REGION Network 4: Block description — Section 3.5 to 3.5
   // ▂▂▂▂▂▂▂▂▂▂▂▂▂▂▂▂▂▂▂▂▂▂▂▂▂▂▂▂▂▂▂▂▂▂▂▂▂▂▂▂▂▂▂▂
   // 3.5     Expressing the calculations in Controller operations
   // 
   // The calculations above must be rendered in a form suitable for the Simatic S7-1500 Controller, 
   // using the mathematical operations available to that Controller, these are listed in Table 2.1.
   // 
   // To perform the calculations in the Controller it will be necessary to use partial calculation to 
   // hold separate components of the overall calculation and combine these to produce the final 
   // result. 
   // 
   // The following sections breakdown each of the response calculations into these partial 
   // calculations and demonstrate how these are then combined to provide a final result that is 
   // compatible with the Controller mathematical operations and Controller notations.
   // 
   // 
   // 
   // ▁▁▁▁▁▁▁▁▁▁▁▁▁▁▁▁▁▁▁▁▁▁▁▁▁▁▁▁▁▁▁▁▁▁▁▁▁▁▁▁▁▁▁▁
   // 3.5.1     Over damped, slow response no overshoot             ζ > 1
   // 
   // 
   // CALCULATION:
   // 
   //       ╓   1 ┌   ζ       ┐   - ω [ ζ ─ √(ζ² ─ 1) ]t       1 ┌   ζ       ┐   - ω [ ζ ┼ √(ζ² ─ 1) ]t ╖
   // y(t) = K║x(t) ─ -- │------------------ ┼ 1│ｅ         ┼ -- │------------------ ─ 1│ｅ           ║
   //       ╙   2 └ √(ζ² ─ 1)     ┘            2 └ √(ζ² ─ 1)     ┘            ╜
   // 
   // 
   // 
   // Is rendered into the correct format as follows:
   // 
   // 
   //  cal_01 = SQRT ( SQR (ζ) - 1)         = √(ζ² ─ 1)
   // 
   //                                  ζ
   //  cal_02 = ζ ÷ cal_01              = -----------------
   //                          √(ζ² ─ 1)
   // 
   //  cal_03 = ζ + cal_01              = ζ ┼ √(ζ² ─ 1)
   // 
   //  cal_04 = -1 × ω × t × cal_03           = - ω [ ζ ┼ √(ζ² ─ 1) ]t
   // 
   //                              -ω [ ζ ┼ √(ζ² ─ 1) ]t 
   //  cal_05 = EXP( cal_04 )              =ｅ
   // 
   //  cal_06 = ζ - cal_01               = ζ ─ √(ζ² ─ 1)
   // 
   //  cal_07 = -1 × ω × t × cal_06           = - ω [ ζ ─ √(ζ² ─ 1) ]t
   // 
   //                            -ω [ ζ ─ √(ζ² ─ 1) ]t 
   //  cal_08 = EXP( cal_07 )              =ｅ
   // 
   //                           1 ┌   ζ       ┐
   //  cal_09 = (cal_02 - 1) × 0.5           = -- │------------------ ─ 1│
   //                           2 └ √(ζ² ─ 1)     ┘
   // 
   //                           1 ┌   ζ       ┐
   //  cal_10 = (cal_02 + 1) × 0.5            = -- │------------------ ┼ 1│
   //                           2 └ √(ζ² ─ 1)     ┘
   // 
   //                           1 ┌   ζ       ┐   -ω [ ζ ┼ √(ζ² ─ 1) ]t
   //  cal_11 = cal_09 × cal_05             = -- │------------------ ─ 1│ｅ
   //                           2 └ √(ζ² ─ 1)     ┘
   // 
   //                           1 ┌   ζ       ┐   -ω [ ζ ─ √(ζ² ─ 1) ]t
   //  cal_12 = cal_10 × cal_08             = -- │------------------ ┼ 1│ｅ
   //                           2 └ √(ζ² ─ 1)     ┘
   // 
   //                          ╓   1 ┌   ζ       ┐   - ω [ ζ ─ √(ζ² ─ 1) ]t       1 ┌   ζ       ┐   - ω [ ζ ┼ √(ζ² ─ 1) ]t ╖
   //  cal_13 = INPUT - cal_12 + cal_11        = ║x(t) ─ -- │------------------ ┼ 1│ｅ         ┼ -- │------------------ ─ 1│ｅ           ║
   //                          ╙   2 └ √(ζ² ─ 1)     ┘            2 └ √(ζ² ─ 1)     ┘            ╜
   // 
   //                             ╓   1 ┌   ζ       ┐   - ω [ ζ ─ √(ζ² ─ 1) ]t       1 ┌   ζ       ┐   - ω [ ζ ┼ √(ζ² ─ 1) ]t ╖
   //  OUTPUT  = K × cal_13             =  K║x(t) ─ -- │------------------ ┼ 1│ｅ         ┼ -- │------------------ ─ 1│ｅ           ║
   //                             ╙   2 └ √(ζ² ─ 1)     ┘            2 └ √(ζ² ─ 1)     ┘            ╜
   // 
   // 
   // 
   // ▁▁▁▁▁▁▁▁▁▁▁▁▁▁▁▁▁▁▁▁▁▁▁▁▁▁▁▁▁▁▁▁▁▁▁▁▁▁▁▁▁▁▁▁
   // 3.5.2     Critically damped, fastest response without overshoot        ζ = 1
   // 
   // 
   // CALCULATION:
   // 
   //       ╓           - ωt  ╖
   // y(t) = K║x(t) ─ (1 ┼ ωt) ｅ  ║
   //       ╙             ╜
   // 
   // 
   // Is rendered into the correct format as follows:
   // 
   // 
   //  cal_01 = -1 × ω × t                = - ωt  
   // 
   //                          - ωt
   //  cal_02 = EXP( cal_01 )              =ｅ
   // 
   //  cal_03 = 1 - cal_01              = 1 ─ (-ωt) = 1 ┼ ωt
   // 
   //                              - ωt
   //  cal_04 = cal_03 × cal_02            = (1 ┼ ωt) ｅ
   // 
   //                                 - ωt
   //  cal_05 = INPUT  - cal_04            = x(t) ─ (1 ┼ ωt) ｅ
   // 
   //                             ╓           - ωt  ╖
   //  OUTPUT  = K × cal_05             =  K║x(t) ─ (1 ┼ ωt) ｅ  ║
   //                             ╙             ╜
   // 
   // 
   // 
   // ▁▁▁▁▁▁▁▁▁▁▁▁▁▁▁▁▁▁▁▁▁▁▁▁▁▁▁▁▁▁▁▁▁▁▁▁▁▁▁▁▁▁▁▁
   // 3.5.3     Under damped, decreasing oscillations              0 < ζ < 1
   // 
   // 
   // CALCULATION:
   // 
   //       ╓      - ζω t  ┌        ζ            ┐╖
   // y(t) = K║x(t) ─ ｅ   │COS (Ωt) ┼ ------------------ SIN (Ωt)│║  where Ω =  ω √(1 ─ ζ²)
   //       ╙       └       √(1 ─ ζ²)       ┘╜
   // 
   // 
   // Is rendered into the correct format as follows:
   // 
   // 
   //  cal_01 = SQRT ( 1 - SQR (ζ))         = √(1 ─ ζ²)
   // 
   //                                  ζ
   //  cal_02 = ζ ÷ cal_01              = -----------------
   //                          √(1 ─ ζ²)
   // 
   //  cal_03 = ω × cal_01                = ω √(1 ─ ζ²) = Ω
   // 
   //  cal_04 = t × cal_03              = Ωt
   // 
   //  cal_05 = COS( cal_04 )             = COS (Ωt)
   // 
   //  cal_06 = SIN( cal_04 )               = SIN (Ωt)
   // 
   //  cal_07 = -1 × ζ × ω × t             = - ζω t 
   // 
   //                          - ζω t 
   //  cal_08 = EXP( cal_07 )              =ｅ
   // 
   //                          - ζω t 
   //  cal_09 = cal_08 × cal_05            =ｅ         COS (Ωt)
   // 
   //  
   //                                  ζ      - ζω t
   //  cal_10 = cal_02 × cal_08 × cal_06        = ----------------- ｅ         SIN (Ωt)
   //                          √(1 ─ ζ²)
   // 
   //                            ╓      - ζω t          ζ     - ζω t            ╖  ╓      - ζω t  ┌        ζ            ┐╖
   //  cal_11 = INPUT - cal_09 - cal_10          =║x(t) ─ ｅ   COS (Ωt) ─ ------------------ ｅ   SIN (Ωt)║=║x(t) ─ ｅ   │COS (Ωt) ┼ ------------------ SIN (Ωt)│║
   //                            ╙              √(1 ─ ζ²)              ╜  ╙       └       √(1 ─ ζ²)       ┘╜
   // 
   //                             ╓      - ζω t  ┌        ζ            ┐╖
   //  OUTPUT  = K × cal_11             =  K║x(t) ─ ｅ   │COS (Ωt) ┼ ------------------ SIN (Ωt)│║
   //                             ╙       └       √(1 ─ ζ²)       ┘╜
   // 
   // 
   // 
   // ▁▁▁▁▁▁▁▁▁▁▁▁▁▁▁▁▁▁▁▁▁▁▁▁▁▁▁▁▁▁▁▁▁▁▁▁▁▁▁▁▁▁▁▁
   // 3.5.4     Undamped, oscillates with frequency ω              ζ = 0
   // 
   // 
   // CALCULATION:
   // 
   //       ╓       ╖
   // y(t) = K║x(t) ─ COS (ωt) ║
   //       ╙       ╜
   // 
   // 
   // Is rendered into the correct format as follows:
   // 
   // 
   //  cal_01 = ω × t                  = ωt
   // 
   //  cal_02 = COS( cal_01 )             = COS (ωt)
   // 
   //  cal_03 = INPUT - cal_02             = x(t) ─ COS (ωt) 
   // 
   //  OUTPUT  = K × cal_03             =  K [ x(t) ─ COS (ωt) ]
   // 
   // 
   // 
   // ▁▁▁▁▁▁▁▁▁▁▁▁▁▁▁▁▁▁▁▁▁▁▁▁▁▁▁▁▁▁▁▁▁▁▁▁▁▁▁▁▁▁▁▁
   // 3.5.5     Unstable, oscillations of increasing amplitude           -1 < ζ < 0
   // 
   // 
   // CALCULATION:
   // 
   //       ╓      | ζ | ω t ┌        ζ            ┐╖
   // y(t) = K║x(t) ─ ｅ    │COS (Ωt) ┼ ------------------ SIN (Ωt)│║  where Ω =  ω √(1 ─ ζ²)
   //       ╙          └       √(1 ─ ζ²)       ┘╜
   // 
   // 
   // Is rendered into the correct format as follows:
   // 
   // 
   //  cal_01 = SQRT ( 1 - SQR (ζ))         = √(1 ─ ζ²)
   // 
   //                                  ζ
   //  cal_02 = ζ ÷ cal_01              = -----------------
   //                          √(1 ─ ζ²)
   // 
   //  cal_03 = ω × cal_01                = ω √(1 ─ ζ²) = Ω
   // 
   //  cal_04 = t × cal_03              = Ωt
   // 
   //  cal_05 = COS( cal_04 )             = COS (Ωt)
   // 
   //  cal_06 = SIN( cal_04 )               = SIN (Ωt)
   // 
   //  cal_07 = ABS(ζ) × ω × t              =  | ζ | ω t 
   // 
   //                           | ζ | ω t 
   //  cal_08 = EXP( cal_07 )              =ｅ
   // 
   //                           | ζ | ω t 
   //  cal_09 = cal_08 × cal_05            =ｅ         COS (Ωt)
   // 
   //  
   //                                  ζ      | ζ | ω t
   //  cal_10 = cal_02 × cal_08 × cal_06        = ----------------- ｅ         SIN (Ωt)
   //                          √(1 ─ ζ²)
   // 
   //                            ╓       | ζ | ω t         ζ      | ζ | ω t         ╖  ╓      | ζ | ω t ┌        ζ            ┐╖
   //  cal_11 = INPUT - cal_09 - cal_10          =║x(t) ─ ｅ   COS (Ωt) ─ ------------------ ｅ   SIN (Ωt)║=║x(t) ─ ｅ    │COS (Ωt) ┼ ------------------ SIN (Ωt)│║
   //                            ╙              √(1 ─ ζ²)              ╜  ╙        └       √(1 ─ ζ²)       ┘╜
   // 
   //                             ╓      | ζ | ω t ┌        ζ            ┐╖
   //  OUTPUT  = K × cal_11             =  K║x(t) ─ ｅ    │COS (Ωt) ┼ ------------------ SIN (Ωt)│║
   //                             ╙          └       √(1 ─ ζ²)       ┘╜
   // 
   // 
   // 
   // ▁▁▁▁▁▁▁▁▁▁▁▁▁▁▁▁▁▁▁▁▁▁▁▁▁▁▁▁▁▁▁▁▁▁▁▁▁▁▁▁▁▁▁▁
   // 3.5.6     Unstable, unbounded asymptotic increase              ζ ≤ -1
   // 
   // 
   // CALCULATION:
   // 
   //       ╓   1 ┌   ζ       ┐     ω [ | ζ | ─ √(ζ² ─ 1) ]t    1 ┌   ζ       ┐     ω [ | ζ | ┼ √(ζ² ─ 1) ]t ╖
   // y(t) = K║x(t) ─ -- │------------------ ┼ 1│ｅ         ┼ -- │------------------ ┼ 1│ｅ              ║
   //       ╙   2 └ √(ζ² ─ 1)     ┘            2 └ √(ζ² ─ 1)     ┘               ╜
   // 
   // 
   // 
   // Is rendered into the correct format as follows:
   // 
   // 
   //  cal_01 = SQRT ( SQR (ζ) - 1)         = √(ζ² ─ 1)
   // 
   //                                  ζ
   //  cal_02 = ζ ÷ cal_01              = -----------------
   //                          √(ζ² ─ 1)
   // 
   //  cal_03 = ABS (ζ) + cal_01            = | ζ | ┼ √(ζ² ─ 1)
   // 
   //  cal_04 = ω × t × cal_03             = ω [ | ζ | ┼ √(ζ² ─ 1) ]t
   // 
   //                               ω [ | ζ | ┼ √(ζ² ─ 1) ]t 
   //  cal_05 = EXP( cal_04 )              =ｅ
   // 
   //  cal_06 = ABS (ζ) - cal_01             =  | ζ | ─ √(ζ² ─ 1)
   // 
   //  cal_07 = ω × t × cal_06             = ω [  | ζ | ─ √(ζ² ─ 1) ]t
   // 
   //                               ω [  | ζ | ─ √(ζ² ─ 1) ]t 
   //  cal_08 = EXP( cal_07 )              =ｅ
   // 
   //                           1 ┌   ζ       ┐
   //  cal_09 = (cal_02 + 1) × 0.5            = -- │------------------ ┼ 1│
   //                           2 └ √(ζ² ─ 1)     ┘
   // 
   //                           1 ┌   ζ       ┐   -ω [ ζ ─ √(ζ² ─ 1) ]t
   //  cal_10 = cal_09 × cal_08             = -- │------------------ ┼ 1│ｅ
   //                           2 └ √(ζ² ─ 1)     ┘
   // 
   //                           1 ┌   ζ       ┐   -ω [ ζ ┼ √(ζ² ─ 1) ]t
   //  cal_11 = cal_09 × cal_05             = -- │------------------ ┼ 1│ｅ
   //                           2 └ √(ζ² ─ 1)     ┘
   // 
   //                          ╓   1 ┌   ζ       ┐   - ω [ ζ ─ √(ζ² ─ 1) ]t       1 ┌   ζ       ┐   - ω [ ζ ┼ √(ζ² ─ 1) ]t ╖
   //  cal_12 = INPUT - cal_10 + cal_11        = ║x(t) ─ -- │------------------ ┼ 1│ｅ         ┼ -- │------------------ ┼ 1│ｅ           ║
   //                          ╙   2 └ √(ζ² ─ 1)     ┘            2 └ √(ζ² ─ 1)     ┘            ╜
   // 
   //                             ╓   1 ┌   ζ       ┐   - ω [ ζ ─ √(ζ² ─ 1) ]t       1 ┌   ζ       ┐   - ω [ ζ ┼ √(ζ² ─ 1) ]t ╖
   //  OUTPUT  = K × cal_12             =  K║x(t) ─ -- │------------------ ┼ 1│ｅ         ┼ -- │------------------ ┼ 1│ｅ           ║
   //                             ╙   2 └ √(ζ² ─ 1)     ┘            2 └ √(ζ² ─ 1)     ┘            ╜
   // 
   // 
   // 
   // ▂▂▂▂▂▂▂▂▂▂▂▂▂▂▂▂▂▂▂▂▂▂▂▂▂▂▂▂▂▂▂▂▂▂▂▂▂▂▂▂▂▂▂▂
   // 3.6     Operating modes
   // 
   // 
   // This block FC19152_StdDebugInst2Order supports manual and automatic operating modes, the 
   // default mode is automatic.
   // 
   // The module can be switched between automatic and manual modes with the 
   // mode_AutMan signal:
   // 
   //  DATA STRUCTURE    UT39152_Dy_DebugInst2Order
   //  ――――――――――――――――――――――――――――――――――――――――――
   //  SIGNAL         FUNCTION               TYPE     DETAILS
   //  ――――――――――――――――――――――――――――――――――――――――――
   //  Mode_AutMan     Specifies the operating mode of     Bool  1 = automatic mode
   //            the simulation                 0 = manual mode
   // 
   //  Mode_Time       Specifies the manual time value of       Real     Elapsed time
   //            the simulation in seconds           in seconds
   // 
   //  status_Aut      The simulation is in automatic mode   Bool  1 = auto mode
   //                                  0 = no in auto
   // 
   //  status_Man       The simulation is in manual mode    Bool  1 = manual mode
   //                                  0 = no in manual
   //  ――――――――――――――――――――――――――――――――――――――――――  
   // 
   // 
   // 
   // ▁▁▁▁▁▁▁▁▁▁▁▁▁▁▁▁▁▁▁▁▁▁▁▁▁▁▁▁▁▁▁▁▁▁▁▁▁▁▁▁▁▁▁▁
   // 3.6.1    Automatic mode
   // 
   // 
   // By default the module will be in automatic mode. 
   // 
   // In automatic mode, if the simulation is active (TRIGGER = 1), the module carries out the relevant 
   // calculation (listed in § 3.2) depending on the value of the damping factor (k_DampFactor) each 
   // time the module is called. The module calculates the elapsed time based on the current CPU 
   // time when the module was called, compared with the CPU time when the simulation was 
   // started (rising edge of TRIGGER) and stored in actual_StartTime.
   // 
   // In automatic mode, a real time simulation occurs, generating responses similar to those shown 
   // in the plots of § 2.3.  
   // 
   // 
   // 
   // ▁▁▁▁▁▁▁▁▁▁▁▁▁▁▁▁▁▁▁▁▁▁▁▁▁▁▁▁▁▁▁▁▁▁▁▁▁▁▁▁▁▁▁▁
   // 3.6.2    Manual mode
   // 
   // 
   // In manual mode, if the simulation is active (TRIGGER = 1), the module carries out the relevant 
   // calculation (listed in § 3.2) depending on the value of the damping factor (k_DampFactor) each 
   // time the module is called; in exactly the same way as automatic mode.
   // 
   // The difference with manual mode, is that the time used in the calculation must be uniquely 
   // specified, the elapsed time is not calculated and a manual time value must be provided.
   // 
   // The manual time is given in the variable mode_ManTime and is specified in seconds.
   // 
   // If mode mode_ManTime remains constant between module calls, the module will return the 
   // same OUTPUT value each time (assuming all other signals remain unchanged).
   // 
   // Manual mode allows the module to calculate the correct response for a particular and exact time, 
   // and is not dependent on cycle times or other factors that may affect when the module is called.
   // 
   // 
   // 
   // ▁▁▁▁▁▁▁▁▁▁▁▁▁▁▁▁▁▁▁▁▁▁▁▁▁▁▁▁▁▁▁▁▁▁▁▁▁▁▁▁▁▁▁▁
   // 3.7      Symbols, block icons and faceplates
   // 
   // There is no supervisory system interface for this block. It is a debug simulation module and as
   // such has no  graphical symbol, block icon or faceplate.
   // 
   //                ━━━   ⬙⬙⬙⬙⬙⬙   ━━━
END_REGION

REGION Network 5: Block description — Sections 4 to 11
   // ▄▄▄▄▄▄▄▄▄▄▄▄▄▄▄▄▄▄▄▄▄▄▄▄▄▄▄▄▄▄▄▄▄▄▄▄▄▄▄▄▄▄▄▄
   // 4.     PARAMETERS
   // 
   // 
   // The following parameters are associated with the block:
   // 
   //  
   //  ――――――――――――――――――――――――――――――――――――――――――
   //  PARAM         FUNCTION                    TYPE      IN-OUT 
   //  ――――――――――――――――――――――――――――――――――――――――――
   //  SYS_SIGNALS      Common system signals              UT21000    In
   //           logic and timing signals for parametric access
   // 
   //  TRIGGER       Activates the simulation (the simulation will run     Bool      In
   //           whilever this signal is high), the elapsed time 
   //           is measured from the rising edge of this signal
   // 
   //  INPUT        The input time function, x(t) in the calculations     Real      In
   // 
   //  DYNAMIC_DATA      Data structure that holds the live data for the       UT39152    InOut
   //           simulation (damping factor, natural frequency, 
   //           system gain, elapsed time &c.)
   // 
   //  OUTPUT       The output time response, y(t) in the calculations   Real      Out
   //  ――――――――――――――――――――――――――――――――――――――――――
   // 
   //                ━━━   ⬙⬙⬙⬙⬙⬙   ━━━
   // 
   // 
   // 
   // ▄▄▄▄▄▄▄▄▄▄▄▄▄▄▄▄▄▄▄▄▄▄▄▄▄▄▄▄▄▄▄▄▄▄▄▄▄▄▄▄▄▄▄▄
   // 5.     DATA STRUCTURES AND USAGE (AND INSTANCE DATA BLOCKS)
   // 
   // 
   // The block has the following associated data structure:
   // 
   // 
   //  ――――――――――――――――――――――――――――――――――――――――――
   //  DATA STRUCTURE             DESCRIPTION
   //  ――――――――――――――――――――――――――――――――――――――――――
   //  UT01000_St_SysRevision          Revision information for this block    See FC01001
   //  UT01001_St_SysLicence           Licence information for this block  See FC01001
   //  UT21000_Dy_SysSignals           System signals for logic and timing  See FC01001
   // 
   //  UT39152_Dy_DebugInst2Orderl       Dynamic data storage, contains live data, such as 
   //                     calculation variables, elapsed time, oscillation 
   //                     frequency and status signals
   //  ――――――――――――――――――――――――――――――――――――――――――
   // 
   // 
   // ▂▂▂▂▂▂▂▂▂▂▂▂▂▂▂▂▂▂▂▂▂▂▂▂▂▂▂▂▂▂▂▂▂▂▂▂▂▂▂▂▂▂▂▂
   // 5.2      UT39152_Dy_DebugInst2Order
   // 
   // The static data structure for an isolating valve.
   // 
   // 
   // 
   //  UT39152_Dy_DebugInst2Order (full contents)
   //  ――――――――――――――――――――――――――――――――――――――――――
   //  SIGNAL NAME          FUNCTION                     TYPE
   //  ――――――――――――――――――――――――――――――――――――――――――
   //  k_Gain             CONSTANT — Simulation system gain        Real
   //  k_NatFreq          CONSTANT — Simulation natural frequency (rad/s)   Real
   //  k_DampFactor        CONSTANT — Simulation damping factor        Real
   //  status_Running      STATUS — Simulation is running  Bool
   //                      (1 = running, 0 = stopped)
   //  status_Stopped        STATUS — Simulation is stopped (not running)    Bool
   //                      (1 = stopped, 0 = running)
   //  status_Stable         STATUS — Simulation response type is stable     Bool
   //                      (1 = stable, 0 = unstable)
   //  status_OverDamp       STATUS — Response is stable/over damped      Bool
   //                      (1 = stable, over damped)
   //  status_CritDamp       STATUS — Response is stable/critically damped     Bool
   //                      (1 = stable, critically damped)
   //  status_UnderDamp     STATUS — Response is stable/under damped      Bool
   //                      (1 = stable, under damped)
   //  status_Undamped      STATUS — Response is stable/undamped       Bool
   //                      (1 = stable, undamped)
   //  status_USUnder        STATUS — Response is unstable/under damped    Bool
   //                      (1 = unstable, under damped)
   //  status_USOver       STATUS — Response is unstable/over damped    Bool
   //                      (1 = unstable, over damped)
   //  status_Osc          STATUS — Oscillatory response             Real
   //                      (1 = osc. response, 0 = non-osc.)
   //  status_OscFreqRS       STATUS — Frequency of oscillation, zero if       Real
   //                      non-oscillatory (rad/s)
   //  status_OscFreqHz       STATUS — Frequency of oscillation, zero if       Real
   //                      non-oscillatory (Hz)
   //  status_Period         STATUS — Period of oscillation, zero if           Real
   //                      non-oscillatory (s)
   //  status_Aut           STATUS — Simulation is in automatic mode      Bool
   //                      (1 = automatic, 0 = manual)
   //  status_Man          STATUS — Simulation is in manual mode        Bool
   //                      (1 = manual, 0 = automatic)
   //  cal_PeakValue          CALC — Peak output value             Real
   //  cal_NatPeriod        CALC — Period of natural oscillations (s)       Real
   //                    zero for non-oscillatory response
   //  cal_DampFreq       CALC — Damped frequency of the system (rad/s)    Real
   //  cal_DampFreqHz         CALC — Damped frequency of the system (Hz)     Real
   //  cal_DampPeriod       CALC — Period of damped oscillations (s)       Real
   //                    zero for non-oscillatory response
   //  cal_TimeSteady        CALC — Time to reach steady state (s)       Real
   //                    zero for unstable response
   //  cal_Time63%          CALC — Time to reach 63% of steady state (s)      Real
   //                    zero for unstable response
   //  cal_TimePeak            CALC — Time to reach the peak ouptut value (s)    Real
   //  mode_AutMan       MODE — Automatic/manual mode selection     Bool
   //                      (1 = auto mode, 0 = manual mode)
   //  mode_ManTime       MODE — Manual mode time value (s)        Real
   //  actual_StartTime         ACTUAL — CPU time when simulation started       Real
   //  actual_RunTime        ACTUAL — Elapsed time since the            Real
   //                      simulation started (s)
   //  ――――――――――――――――――――――――――――――――――――――――――
   // 
   // 
   //                ━━━   ⬙⬙⬙⬙⬙⬙   ━━━
   // 
   // 
   // 
   // ▄▄▄▄▄▄▄▄▄▄▄▄▄▄▄▄▄▄▄▄▄▄▄▄▄▄▄▄▄▄▄▄▄▄▄▄▄▄▄▄▄▄▄▄
   // 6.     CONSTANTS AND TEMPORARY (LOCAL) DATA
   // 
   // There is no constant data.
   // 
   // The following temporary data is used:
   // 
   //  Temporary (local) data
   //  ――――――――――――――――――――――――――――――――――――――――――
   //  SIGNAL NAME          FUNCTION                  TYPE
   //  ――――――――――――――――――――――――――――――――――――――――――
   //  revInfo             Revision information for the block         UT01000
   //  licInfo           Licensing information for the block      UT01001
   //  cal_01          Partial calculation see § 3.5 for details      Real
   //  cal_02          Partial calculation see § 3.5 for details      Real
   //  cal_03          Partial calculation see § 3.5 for details      Real
   //  cal_04          Partial calculation see § 3.5 for details      Real
   //  cal_05          Partial calculation see § 3.5 for details      Real
   //  cal_06          Partial calculation see § 3.5 for details      Real
   //  cal_07          Partial calculation see § 3.5 for details      Real
   //  cal_08          Partial calculation see § 3.5 for details      Real
   //  cal_09          Partial calculation see § 3.5 for details      Real
   //  cal_10          Partial calculation see § 3.5 for details      Real
   //  cal_11          Partial calculation see § 3.5 for details      Real
   //  cal_12          Partial calculation see § 3.5 for details      Real
   //  cal_13          Partial calculation see § 3.5 for details      Real
   //  wrkInt           Working storage area (integer)          Int
   //  wrkDInt           Working storage area (double integer)         DInt
   //  wrkLInt            Working storage area (long integer)        LInt
   //  wrkLTime           Working storage area (long time)         LT
   //  wrkDTL            Working storage area (DateTime long)      DTL
   //  wrkReal           Working storage (Real)             Real
   //  ―――――――――――――――――――――――――――――――――――――――――― █ █ █
   // 
   //                ━━━   ⬙⬙⬙⬙⬙⬙   ━━━
   // 
   // 
   // 
   // ▄▄▄▄▄▄▄▄▄▄▄▄▄▄▄▄▄▄▄▄▄▄▄▄▄▄▄▄▄▄▄▄▄▄▄▄▄▄▄▄▄▄▄▄
   // 7.     BLOCK CALLS
   // 
   // There are no PAL block calls from within this block.
   // 
   //                ━━━   ⬙⬙⬙⬙⬙⬙   ━━━
   // 
   // 
   // 
   // ▄▄▄▄▄▄▄▄▄▄▄▄▄▄▄▄▄▄▄▄▄▄▄▄▄▄▄▄▄▄▄▄▄▄▄▄▄▄▄▄▄▄▄▄
   // 8.     ASSOCIATED BLOCKS
   // 
   // 
   // This is a stand-alone block and is not associated with any other blocks.
   // 
   //                ━━━   ⬙⬙⬙⬙⬙⬙   ━━━
   // 
   // 
   // 
   // ▄▄▄▄▄▄▄▄▄▄▄▄▄▄▄▄▄▄▄▄▄▄▄▄▄▄▄▄▄▄▄▄▄▄▄▄▄▄▄▄▄▄▄▄
   // 9.     SYSTEM BLOCK CALLS AND SYSTEM DATA TYPES
   // 
   // The following calls are made to system blocks:
   // 
   // 
   //  System block calls
   //  ――――――――――――――――――――――――――――――――――――――――――
   //  BLOCK          TITLE             DESCRIPTION  
   //  ――――――――――――――――――――――――――――――――――――――――――
   //  RD_LOC_T             Read the local RTC time    Reads the CPU real time clock 
   //  ――――――――――――――――――――――――――――――――――――――――――
   // 
   // There are no special system data types used.
   // 
   // 
   //                ━━━   ⬙⬙⬙⬙⬙⬙   ━━━
   // 
   // 
   // 
   // ▄▄▄▄▄▄▄▄▄▄▄▄▄▄▄▄▄▄▄▄▄▄▄▄▄▄▄▄▄▄▄▄▄▄▄▄▄▄▄▄▄▄▄▄
   // 10.     SPECIAL PROPERTIES AND REQUIREMENTS
   // 
   // 
   // 
   // ▂▂▂▂▂▂▂▂▂▂▂▂▂▂▂▂▂▂▂▂▂▂▂▂▂▂▂▂▂▂▂▂▂▂▂▂▂▂▂▂▂▂▂▂
   // 10.1   Block optimisation
   // 
   // 
   // Block optimisation is ACTIVE for this block
   // 
   // 
   // 
   // ▂▂▂▂▂▂▂▂▂▂▂▂▂▂▂▂▂▂▂▂▂▂▂▂▂▂▂▂▂▂▂▂▂▂▂▂▂▂▂▂▂▂▂▂
   // 10.2   Calling requirements
   // 
   // 
   // There are no special calling requirements for this block.
   // 
   //                ━━━   ⬙⬙⬙⬙⬙⬙   ━━━
   // 
   // 
   // 
   // ▄▄▄▄▄▄▄▄▄▄▄▄▄▄▄▄▄▄▄▄▄▄▄▄▄▄▄▄▄▄▄▄▄▄▄▄▄▄▄▄▄▄▄▄
   // 11.     EXAMPLE USAGE
   // 
   // 
   // The following shows a typical deployment of FC19512:
   // 
   //                         ┌─────────────
   //      ───────────────────┤ FC19512
   //                         ├───────────────┤
   //    "DB21001_DY_StdGlobalData".SysSignals ─┤ SYS_SIGNALS            
   //                         │               OUTPUT ├─  "wrk_Real"
   //                         │               │
   //                                                        "1.0" ─┤ INPUT                     │
   //                         │               │
   //                   %M999.0     │               │
   //                    "SIM01_TRIG" ─┤ TRIGGER                     │
   //                         │               │
   //                         │
   //       "DB39152_Dy_DebugInst2Order".S001 ─┤ DYNAMIC_DATA
   //                         │
   //                         │
   //                                         │
   //                                ─────────┘
   // 
   // 
   //               ━━━   ⬙⬙⬙⬙⬙⬙   ━━━
   // 
   // 
   // ██████████████ █ █ █ █  END   █ █ █ █ ██████████████
END_REGION

REGION Network 6: Current revision and modification history
   // ▄▄▄▄▄▄▄▄▄▄▄▄▄▄▄▄▄▄▄▄▄▄▄▄▄▄▄▄▄▄▄▄▄▄▄▄▄▄▄▄▄▄▄▄
   // MODIFICATION HISTORY
   // 
   // 
   // The revision data shown here, in the network comments, contains additional information 
   // reflecting the software development workflow under the version control system (VCS) employed 
   // to track all software changes.
   // 
   // The VCS in use is the Git Source Code Management system in conjunction with the GitHub online 
   // hosting system. The software in its entirety is available in the GitHub remote repository:
   // 
   //      https://github.com/practicalseries/PS2001-pal-software
   // 
   // The repository is public and can be freely copied (forked in GitHub terminology) and used 
   // under the MIT licence. 
   // 
   // The MIT licence is reproduced in full in the last network of this software module.
   // 
   // 
   //  ―――――――――――――――――――――――――――――――――――――――――――
   //  DATE       REVISION             MASTER BRANCH     DEV
   //          (nnn.amm)   COMMIT TAG    (Base ---> Merge)    BRANCH   Author
   //  ———————————————————————————————————————————
   //  2022.01.12    000.101   D0009A-000.101   D0009 N/A     D0009A   M. Gledhill
   //                        FC19512 Block created — Comments added
   //  ———————————————————————————————————————————
   //   Where: nnn  =  Major revision
   //         a  =  Type (1-7 Development, 8 Proving, 9 Qualification, 0 Release)
   //       mm  =  Minor revision (must be 00 if a = 0)
   //         Block properties version number should be set to nn.a (only one decimal place)
   // 
   // ▄▄▄▄▄▄▄▄▄▄▄▄▄▄▄▄▄▄▄▄▄▄▄▄▄▄▄▄▄▄▄▄▄▄▄▄▄▄▄▄▄▄▄▄
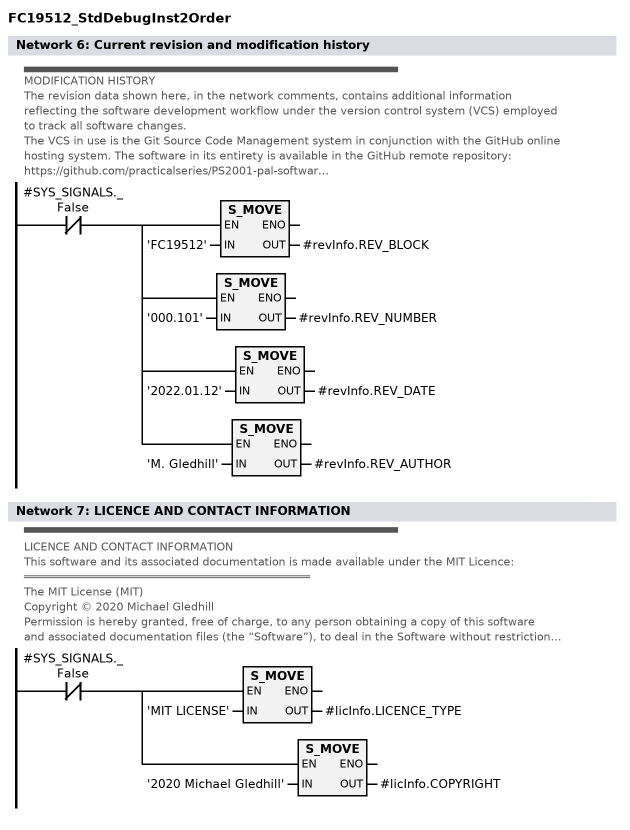
   RUNG wire#powerrail
      I_Contact( #SYS_SIGNALS._False )
      wire#w1
      S_Move(in := 'FC19512', out => #revInfo.REV_BLOCK)
   END_RUNG
   RUNG wire#w1
      S_Move(in := '000.101', out => #revInfo.REV_NUMBER)
   END_RUNG
   RUNG wire#w1
      S_Move(in := '2022.01.12', out => #revInfo.REV_DATE)
   END_RUNG
   RUNG wire#w1
      S_Move(in := 'M. Gledhill', out => #revInfo.REV_AUTHOR)
   END_RUNG
   // the same network as SCL:
   IF NOT #SYS_SIGNALS._False THEN
       #revInfo.REV_BLOCK := 'FC19512';
       #revInfo.REV_NUMBER := '000.101';
       #revInfo.REV_DATE := '2022.01.12';
       #revInfo.REV_AUTHOR := 'M. Gledhill';
   END_IF;
END_REGION

REGION Network 7: LICENCE AND CONTACT INFORMATION
   // ▀▀▀▀▀▀▀▀▀▀▀▀▀▀▀▀▀▀▀▀▀▀▀▀▀▀▀▀▀▀▀▀▀▀▀▀▀▀▀▀▀▀▀▀
   // LICENCE AND CONTACT INFORMATION
   // 
   // This software and its associated documentation is made available under the MIT Licence:
   // 
   // ════════════════════════════════════════════
   // 
   // The MIT License (MIT)
   // 
   // Copyright © 2020 Michael Gledhill
   // 
   // Permission is hereby granted, free of charge, to any person obtaining a copy of this software 
   // and associated documentation files (the “Software”), to deal in the Software without restriction, 
   // including without limitation the rights to use, copy, modify, merge, publish, distribute, 
   // sublicense, and/or sell copies of the Software, and to permit persons to whom the Software is 
   // furnished to do so, subject to the following conditions: 
   // 
   // The above copyright notice and this permission notice shall be included in all copies or 
   // substantial portions of the Software.
   // 
   // THE SOFTWARE IS PROVIDED “AS IS”, WITHOUT WARRANTY OF ANY KIND, EXPRESS OR IMPLIED, 
   // INCLUDING BUT NOT LIMITED TO THE WARRANTIES OF MERCHANTABILITY, FITNESS FOR A 
   // PARTICULAR PURPOSE AND NON-INFRINGEMENT. IN NO EVENT SHALL THE AUTHORS OR COPYRIGHT 
   // HOLDERS BE LIABLE FOR ANY CLAIM, DAMAGES OR OTHER LIABILITY, WHETHER IN AN ACTION OF 
   // CONTRACT, TORT OR OTHERWISE, ARISING FROM, OUT OF OR IN CONNECTION WITH THE SOFTWARE 
   // OR THE USE OR OTHER DEALINGS IN THE SOFTWARE.
   // 
   // ════════════════════════════════════════════
   //                    ┌────────────┐
   // You can reach the author by email here:   │  mg@practicalseries.com  │
   //                    └────────────┘
   // Questions, corrections, constructive criticism and complaints (polite ones) are invited.
   RUNG wire#powerrail
      I_Contact( #SYS_SIGNALS._False )
      wire#w1
      S_Move(in := 'MIT LICENSE', out => #licInfo.LICENCE_TYPE)
   END_RUNG
   RUNG wire#w1
      S_Move(in := '2020 Michael Gledhill', out => #licInfo.COPYRIGHT)
   END_RUNG
   // the same network as SCL:
   IF NOT #SYS_SIGNALS._False THEN
       #licInfo.LICENCE_TYPE := 'MIT LICENSE';
       #licInfo.COPYRIGHT := '2020 Michael Gledhill';
   END_IF;
END_REGION
END_FUNCTION

FUNCTION "FC61000_DocGenExample" : Void   // FC61000, LAD
TITLE = Documentation - Gen — Example Documentation (full)
{ S7_Optimized_Access := 'TRUE' }
AUTHOR : M_Gledhill
FAMILY : Documentation
NAME : DocGenExample
VERSION : 1.1
// PRACTICAL SERIES AUTOMATION LIBRARY (PAL)   —   COPYRIGHT 2020 – M. GLEDHILL (MIT LICENCE)
//                   ———— ◆ ————
//  FOR DETAILED DOCUMENTATION — SELECT THE BLOCK IN THE PROJECT TREE AND PRESS SHIFT + F1
//  FULL ONLINE DOCUMENTATION IS AVAILABLE AT: https://practicalseries.com/2001-pal/index.html
// stored: AutoNumber false, IsIECCheckEnabled false, SetENOAutomatically false, UDAEnableTagReadback false
   VAR_INPUT
      SYS_SIGNALS : "UT21000_Dy_SysSignals";   // Common system signals — logic and timing signals
   END_VAR
   VAR_TEMP
      revInfo : "UT01000_St_SysRevision";   // Revision information for this block
      licInfo : "UT01001_St_SysLicence";   // Licence information for this block
      wrkReal : Real;   // Working storage (real)
   END_VAR
BEGIN

REGION Network 1: Block description
   // ▀▀▀▀▀▀▀▀▀▀▀▀▀▀▀▀▀▀▀▀▀▀▀▀▀▀▀▀▀▀▀▀▀▀▀▀▀▀▀▀▀▀▀▀
   // 
   // TITLE:    EXAMPLE DOCUMENTATION FOR USE IN COMMENTS
   // 
   // ▄▄▄▄▄▄▄▄▄▄▄▄▄▄▄▄▄▄▄▄▄▄▄▄▄▄▄▄▄▄▄▄▄▄▄▄▄▄▄▄▄▄▄▄
   // 
   // 
   // 
   // This block contains examples of all the typical forms of documentation used within the PAL
   // software. It provides the following:
   // 
   // CONTENTS (BY NETWORK)
   // 
   // NW 1.    Block Contents
   // NW 2.    Current revision and modification history
   // 
   // 
   // EXAMPLES
   // 
   // NW 3.    Example — Block description — Sections 1 to 3
   // NW 4.    Example — Block description — Sections 4 to 11
   // NW 5.    Example — Current revision and modification history
   // NW 6.    Example — Headings, lists and indented text
   // NW 7.    Example — Body text
   // NW 8.    Example — Standard Tables
   // NW 9.    Example — Other tables
   // NW 10.    Example — Equations
   // NW 11.    Example — Figures
   // 
   // 
   // CHARACTER LISTS
   // 
   // NW 12.    Special characters — Hyphens, whitespace and construction lines
   // NW 13.    Special characters — Arrows, box and block characters
   // NW 14.    Special characters — Currency, punctuation and full-width characters
   // NW 15.    Special characters — Greek, indexing characters and Roman numerals
   // NW 16.    Special characters — Mathematical operators (including vulgar fractions)
   // NW 17.    Special characters — Geometrical and ornamental characters
   // NW 18.    Special characters — Common character widths and additional whitespace characters
   // 
   // 
   // SPECIAL NETWORKS
   // 
   // NW 19.    OB1 NETWORK 1 — Project description
   // NW 20.    OB1 NETWORK 2 — Current revision and modification history
   // 
   // TYPICAL NETWORK COMMENTS
   // 
   // NW 21.    Load the system RTC and store in local variable  [typical network comment]
   // NW 22.    ██ STEP 03340 — DECLARATION (RUNNING)    [sequence network comment]
   // NW 23.       STEP 03340 — ACTION (INITIALISE)           [sequence network comment]
   // NW 24.       STEP 03340 — TRANSITION 01                   [sequence network comment]
   // NW 25.   LICENCE AND CONTACT INFORMATION       [final network]
   // 
   //               ━━━   ⬙⬙⬙⬙⬙⬙   ━━━
   // 
   // 
   // 
   // ▄▄▄▄▄▄▄▄▄▄▄▄▄▄▄▄▄▄▄▄▄▄▄▄▄▄▄▄▄▄▄▄▄▄▄▄▄▄▄▄▄▄▄▄
   // 1.     BLOCK TECHNICAL SUMMARY
   // 
   // 
   //  ――――――――――――――――――――――――――――――――――――――――――
   //  NOMENCLATURE & ADDRESSING
   //  ――――――――――――――――――――――――――――――――――――――――――
   //  BLOCK TITLE         Example Documentation for use in Comments
   //  BLOCK FUNCTION GROUP    Documentation
   //  BLOCK ADDRESS       FC 61000
   //  BLOCK SYMBOL        FC61000_DocGenExample
   //  BLOCK USER ID         DocGenExample
   // 
   //  ――――――――――――――――――――――――――――――――――――――――――
   //  BLOCK TYPE & USAGE
   //  ――――――――――――――――――――――――――――――――――――――――――
   //  BLOCK TYPE         Function (FC)
   //  BLOCK NUMBER        61000
   //  LANGUAGE           LAD
   //  OPTIMISED ACCESS     Yes
   //  PAL USAGE TYPE       Standard block
   // 
   //  ――――――――――――――――――――――――――――――――――――――――――
   //  METRICS
   //  ――――――――――――――――――――――――――――――――――――――――――
   //  EXECUTION TIME       24.48 μs¹
   //  LOAD MEMORY       51.63 kB  (52873 bytes)
   //  WORK MEMORY           0.37 kB      (376 bytes)
   //  ――――――――――――――――――――――――――――――――――――――――――
   //                ¹ Measured on: CPU-1515-2PN (order no. 6ES7 512-2AM02-0AB0)
   // 
   //                ━━━   ⬙⬙⬙⬙⬙⬙   ━━━
   // 
   // 
   // 
   // ▄▄▄▄▄▄▄▄▄▄▄▄▄▄▄▄▄▄▄▄▄▄▄▄▄▄▄▄▄▄▄▄▄▄▄▄▄▄▄▄▄▄▄▄
   // 2.     FUNCTIONAL DESCRIPTION
   // 
   // 
   // FC61000 is a documentation module that contains examples of all the common block and 
   // network comments used throughout the PAL software.
   // 
   // All examples are based upon the Style Guide (Doc. No. PS2001-5-2313-011).
   // 
   // FC61000 also contains lists of the characters available within the Siemens TIA font used within
   // all comment sections.
   // 
   //                ━━━   ⬙⬙⬙⬙⬙⬙   ━━━
   // 
   // 
   // 
   // ▄▄▄▄▄▄▄▄▄▄▄▄▄▄▄▄▄▄▄▄▄▄▄▄▄▄▄▄▄▄▄▄▄▄▄▄▄▄▄▄▄▄▄▄
   // 3.     DETAILED BLOCK DESCRIPTION
   // 
   // 
   // The purpose of this block is to provide an easy point of reference for the various documentation 
   // constructs and styles used within the PAL.
   // 
   // The block itself does not contain any executable code, with the exception of the revision and
   // licence networks, all networks are empty. The block itself does nothing, and its execution will
   // have no effect, other than extending the cycle time.
   // 
   //                ━━━   ⬙⬙⬙⬙⬙⬙   ━━━
   // 
   // 
   // 
   // ▄▄▄▄▄▄▄▄▄▄▄▄▄▄▄▄▄▄▄▄▄▄▄▄▄▄▄▄▄▄▄▄▄▄▄▄▄▄▄▄▄▄▄▄
   // 4.     PARAMETERS
   // 
   // 
   // This block has no parameters.
   // 
   //                ━━━   ⬙⬙⬙⬙⬙⬙   ━━━
   // 
   // 
   // 
   // ▄▄▄▄▄▄▄▄▄▄▄▄▄▄▄▄▄▄▄▄▄▄▄▄▄▄▄▄▄▄▄▄▄▄▄▄▄▄▄▄▄▄▄▄
   // 5.     DATA STRUCTURES AND USAGE (AND INSTANCE DATA BLOCKS)
   // 
   // 
   // The block has the following associated data structure:
   // 
   // 
   //  ――――――――――――――――――――――――――――――――――――――――――
   //  DATA STRUCTURE             DESCRIPTION
   //  ――――――――――――――――――――――――――――――――――――――――――
   //  UT01000_St_SysRevision          Revision information for this block    See FC01001
   //  UT01001_St_SysLicence           Licence information for this block  See FC01001
   //  ――――――――――――――――――――――――――――――――――――――――――
   // 
   // 
   //                ━━━   ⬙⬙⬙⬙⬙⬙   ━━━
   // 
   // 
   // 
   // ▄▄▄▄▄▄▄▄▄▄▄▄▄▄▄▄▄▄▄▄▄▄▄▄▄▄▄▄▄▄▄▄▄▄▄▄▄▄▄▄▄▄▄▄
   // 6.     CONSTANTS AND TEMPORARY (LOCAL) DATA
   // 
   // 
   // The following constants and temporary data storage are used:
   // 
   // 
   //  Temporary (local) data
   //  ――――――――――――――――――――――――――――――――――――――――――
   //  SIGNAL NAME          FUNCTION                  TYPE
   //  ――――――――――――――――――――――――――――――――――――――――――
   //  revInfo             Revision information for the block         UT01000
   //  licInfo           Licensing information for the block      UT01001
   //  wrkReal           Working storage (Real)             Real
   //  ――――――――――――――――――――――――――――――――――――――――――
   // 
   // 
   //  Constants data
   //  ――――――――――――――――――――――――――――――――――――――――――
   //  SIGNAL NAME          FUNCTION                  TYPE
   //  ――――――――――――――――――――――――――――――――――――――――――
   //  _FALSE            Temporary internal "False" signal      Bool
   //  ――――――――――――――――――――――――――――――――――――――――――
   // 
   // 
   //                ━━━   ⬙⬙⬙⬙⬙⬙   ━━━
   // 
   //  
   // 
   // ▄▄▄▄▄▄▄▄▄▄▄▄▄▄▄▄▄▄▄▄▄▄▄▄▄▄▄▄▄▄▄▄▄▄▄▄▄▄▄▄▄▄▄▄
   // 7.     BLOCK CALLS
   // 
   // 
   // There are no PAL block calls from within this block.
   // 
   //                ━━━   ⬙⬙⬙⬙⬙⬙   ━━━
   // 
   // 
   // 
   // ▄▄▄▄▄▄▄▄▄▄▄▄▄▄▄▄▄▄▄▄▄▄▄▄▄▄▄▄▄▄▄▄▄▄▄▄▄▄▄▄▄▄▄▄
   // 8.     ASSOCIATED BLOCKS
   // 
   // 
   // This is a stand-alone block and is not associated with any other blocks.
   // 
   //                ━━━   ⬙⬙⬙⬙⬙⬙   ━━━
   // 
   // 
   // 
   // 9.     SYSTEM BLOCK CALLS AND SYSTEM DATA TYPES
   // 
   // There are no system block calls.
   // 
   //                ━━━   ⬙⬙⬙⬙⬙⬙   ━━━
   // 
   // 
   // 
   // ▄▄▄▄▄▄▄▄▄▄▄▄▄▄▄▄▄▄▄▄▄▄▄▄▄▄▄▄▄▄▄▄▄▄▄▄▄▄▄▄▄▄▄▄
   // 10.     SPECIAL PROPERTIES AND REQUIREMENTS
   // 
   // 
   // 
   // ▂▂▂▂▂▂▂▂▂▂▂▂▂▂▂▂▂▂▂▂▂▂▂▂▂▂▂▂▂▂▂▂▂▂▂▂▂▂▂▂▂▂▂▂
   // 10.1   Block optimisation
   // 
   // 
   // Block optimisation is ACTIVE for this block
   // 
   // 
   // 
   // ▂▂▂▂▂▂▂▂▂▂▂▂▂▂▂▂▂▂▂▂▂▂▂▂▂▂▂▂▂▂▂▂▂▂▂▂▂▂▂▂▂▂▂▂
   // 10.2   Calling requirements
   // 
   // 
   // There are no special calling requirements for this block.
   // 
   //                ━━━   ⬙⬙⬙⬙⬙⬙   ━━━
   // 
   // 
   // 
   // ▄▄▄▄▄▄▄▄▄▄▄▄▄▄▄▄▄▄▄▄▄▄▄▄▄▄▄▄▄▄▄▄▄▄▄▄▄▄▄▄▄▄▄▄
   // 11.     EXAMPLE USAGE
   // 
   // 
   // The following shows a typical deployment of FC61000:
   // 
   // 
   //                        ┌────────────
   //    ────────────────────┤ FC61000 
   //                        ├──────────
   //      "DB21001_DY_StdGlobalData".SysSignals ─┤ SYS_SIGNALS
   //                        │
   //                        │               │
   //                        │               │
   //                                     │
   //                        ─────────────┘
   // 
   //               ━━━   ⬙⬙⬙⬙⬙⬙   ━━━
   // 
   // 
   // ██████████████ █ █ █ █  END   █ █ █ █ ██████████████
END_REGION

REGION Network 2: Current revision and modification history
   // ▄▄▄▄▄▄▄▄▄▄▄▄▄▄▄▄▄▄▄▄▄▄▄▄▄▄▄▄▄▄▄▄▄▄▄▄▄▄▄▄▄▄▄▄
   // MODIFICATION HISTORY
   // 
   // The revision data shown here, in the network comments, contains additional information 
   // reflecting the software development workflow under the version control system (VCS) employed 
   // to track all software changes.
   // 
   // The VCS in use is the Git Source Code Management system in conjunction with the GitHub online 
   // hosting system. The software in its entirety is available in the GitHub remote repository:
   // 
   //      https://github.com/practicalseries/PS2001-pal-software
   // 
   // The repository is public and can be freely copied (forked in GitHub terminology) and used 
   // under the MIT licence. 
   // 
   // The MIT licence is reproduced in full in the last network of this software module.
   // 
   // 
   //  ―――――――――――――――――――――――――――――――――――――――――――
   //  DATE       REVISION             MASTER BRANCH     DEV
   //          (nnn.amm)   COMMIT TAG    (Base ---> Merge)    BRANCH   Author
   //  ———————————————————————————————————————————
   //  2021.08.10    001.102   D0008A-000.103   D0008 N/A     D0008A   M. Gledhill
   //                        Constants table added to network 8
   // 
   //  2021.05.18    001.101   D0005A-000.102   D0005 N/A     D0005A   M. Gledhill
   //                        OB1 secondary commit revision added
   //                        OB1 document list updated
   // 
   //  2021.02.18    001.000   D0002      D0001 D0002  None    M. Gledhill
   //                        FC61000 — RELEASED FOR USE
   //                          Block imported form 000.125-Db
   //  ———————————————————————————————————————————
   //   Where: nnn  =  Major revision
   //         a  =  Type (1-7 Development, 8 Proving, 9 Qualification, 0 Release)
   //       mm  =  Minor revision (must be 00 if a = 0)
   //         Block properties version number should be set to nn.a (only one decimal place)
   // 
   // ▄▄▄▄▄▄▄▄▄▄▄▄▄▄▄▄▄▄▄▄▄▄▄▄▄▄▄▄▄▄▄▄▄▄▄▄▄▄▄▄▄▄▄▄
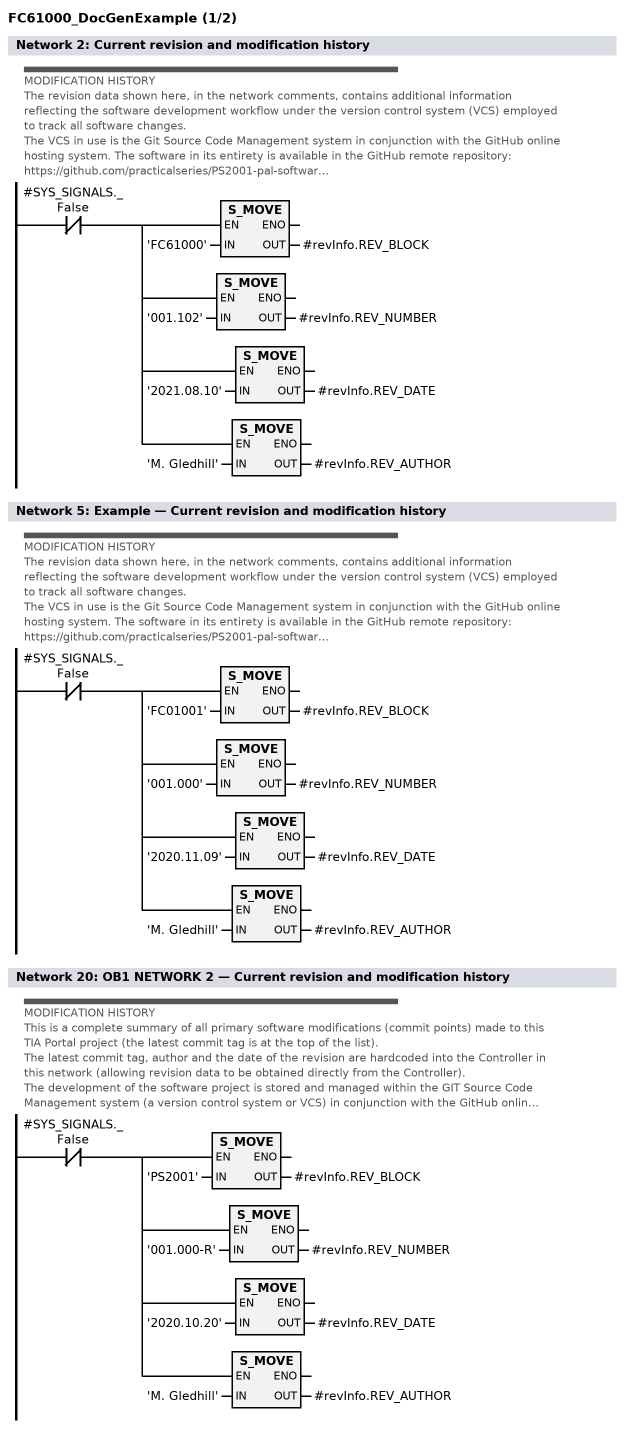
   RUNG wire#powerrail
      I_Contact( #SYS_SIGNALS._False )
      wire#w1
      S_Move(in := 'FC61000', out => #revInfo.REV_BLOCK)
   END_RUNG
   RUNG wire#w1
      S_Move(in := '001.102', out => #revInfo.REV_NUMBER)
   END_RUNG
   RUNG wire#w1
      S_Move(in := '2021.08.10', out => #revInfo.REV_DATE)
   END_RUNG
   RUNG wire#w1
      S_Move(in := 'M. Gledhill', out => #revInfo.REV_AUTHOR)
   END_RUNG
   // the same network as SCL:
   IF NOT #SYS_SIGNALS._False THEN
       #revInfo.REV_BLOCK := 'FC61000';
       #revInfo.REV_NUMBER := '001.102';
       #revInfo.REV_DATE := '2021.08.10';
       #revInfo.REV_AUTHOR := 'M. Gledhill';
   END_IF;
END_REGION

REGION Network 3: Example — Block description — Sections 1 to 3
   // | ▀▀▀▀▀▀▀▀▀▀▀▀▀▀▀▀▀▀▀▀▀▀▀▀▀▀▀▀▀▀▀▀▀▀▀▀▀▀▀▀▀▀▀▀
   // 
   // TITLE:    SUBROUTINE — EVENT TIMER USING RTC
   // 
   // ▄▄▄▄▄▄▄▄▄▄▄▄▄▄▄▄▄▄▄▄▄▄▄▄▄▄▄▄▄▄▄▄▄▄▄▄▄▄▄▄▄▄▄▄
   //  
   // 
   // 
   // This block (FC18151_SubTimeEventRTC) is a subroutine block that times the duration of an event 
   // to nanosecond resolution.
   // 
   // The block records the time the event started (rising edge of the TRIGGER signal), the time the 
   // event ended (falling edge of the TRIGGER signal) and calculates the duration of the event (end 
   // time minus the start time).
   // 
   // The start and end times are read from the real time clock of the controller.
   // 
   // This is a subroutine block.
   // 
   //                ━━━   ⬙⬙⬙⬙⬙⬙   ━━━
   // 
   // 
   // 
   // ▄▄▄▄▄▄▄▄▄▄▄▄▄▄▄▄▄▄▄▄▄▄▄▄▄▄▄▄▄▄▄▄▄▄▄▄▄▄▄▄▄▄▄▄
   // 1.     BLOCK TECHNICAL SUMMARY
   // 
   // 
   //  ――――――――――――――――――――――――――――――――――――――――――
   //  NOMENCLATURE & ADDRESSING
   //  ――――――――――――――――――――――――――――――――――――――――――
   //  BLOCK TITLE         Subroutine Event Timer using RTC
   //  BLOCK FUNCTION GROUP    Subroutine
   //  BLOCK ADDRESS       FC18151
   //  BLOCK SYMBOL        FC18151_SubTimeEventRTC
   //  BLOCK USER ID         SubTimeEventRTC
   // 
   //  ――――――――――――――――――――――――――――――――――――――――――
   //  BLOCK TYPE & USAGE
   //  ――――――――――――――――――――――――――――――――――――――――――
   //  BLOCK TYPE         Function (FC)
   //  BLOCK NUMBER        18151
   //  LANGUAGE           LAD
   //  OPTIMISED ACCESS     Yes
   //  PAL USAGE TYPE       Standard block
   // 
   //  ――――――――――――――――――――――――――――――――――――――――――
   //  METRICS
   //  ――――――――――――――――――――――――――――――――――――――――――
   //  EXECUTION TIME       18.41 μs¹
   //  LOAD MEMORY       23.11 kB  (23667 bytes)
   //  WORK MEMORY           0.43 kB      (442 bytes)
   //  ――――――――――――――――――――――――――――――――――――――――――
   //                ¹ Measured on: CPU-1515-2PN (order no. 6ES7 512-2AM02-0AB0)
   // 
   //                ━━━   ⬙⬙⬙⬙⬙⬙   ━━━
   // 
   // 
   // 
   // ▄▄▄▄▄▄▄▄▄▄▄▄▄▄▄▄▄▄▄▄▄▄▄▄▄▄▄▄▄▄▄▄▄▄▄▄▄▄▄▄▄▄▄▄
   // 2.     FUNCTIONAL DESCRIPTION
   // 
   // 
   // FC18151 is the Subroutine Event Timer using RTC block, it simply records the duration of an event 
   // with a high degree of accuracy. The event being timed is a Boolean signal passed to the block as 
   // the TRIGGER parameter.
   // 
   // Three times are recorded for the event, the start time (rising edge of the TRIGGER parameter), the 
   // end time (falling edge of the TRIGGER parameter) and the duration of the event (end time minus 
   // the start time). The duration is calculated on the falling edge of the TRIGGER parameter, 
   // immediately after the end time is recorded.
   // 
   // The start and end times are read from the Controller’s internal real time clock (RTC) and are 
   // stored in DTL (date time long) format, this format contains year, month, day, hours, minutes, 
   // seconds, milliseconds, microseconds and nano seconds.
   // 
   // The duration is stored in LTime (long time, 64-bit) format, and is very accurate, it resolves to 
   // days, hours, minutes, seconds milliseconds, microseconds and nanoseconds, it keeps this 
   // resolution irrespective of the duration.
   // 
   // The duration is also calculated as a real number in seconds (or fractions thereof); this is a 
   // more convenient format for holding the duration, but is not as accurate as the LTime format.
   // 
   //                ━━━   ⬙⬙⬙⬙⬙⬙   ━━━
   // 
   // 
   // 
   // ▄▄▄▄▄▄▄▄▄▄▄▄▄▄▄▄▄▄▄▄▄▄▄▄▄▄▄▄▄▄▄▄▄▄▄▄▄▄▄▄▄▄▄▄
   // 3.     DETAILED BLOCK DESCRIPTION
   // 
   // 
   // The purpose of this block is to determine with a high degree of accuracy the duration of an event, 
   // the event itself must be in the form of a Boolean trigger signal, the rising edge of the signal is 
   // considered to be the start of the event and the falling edge the end of the event.
   // 
   // The event signal is passed to the block as the TRIGGER parameter. 
   // The block returns five values, these are stored in a UDT passed to the block in the 
   // DYNAMIC_DATA parameter: 
   // 
   // 
   //  ――――――――――――――――――――――――――――――――――――――――――
   //  PARAM         ASSOCIATED UDT            ASSOCIATED DATA BLOCK
   //  ――――――――――――――――――――――――――――――――――――――――――
   //  DYNAMIC_DATA     UT38151_Dy_SubTimeEventRTC       DB38151_Dy_SubTimeEventRTC
   //  ――――――――――――――――――――――――――――――――――――――――――
   // 
   // 
   // The block returns the following data:
   // 
   // 
   //  UT38151_Dy_SubTimeEventRTC
   //  ―――――――――――――――――――――――――――――――――――――――――― 
   //  SIGNAL NAME          FUNCTION                     TYPE
   //  ――――――――――――――――――――――――――――――――――――――――――
   //  status_Running      STATUS — The event timer is running         Bool
   // 
   //  actual_StartTime      ACTUAL — Time at which the TRIGGER signal        DTL
   //                      went high (event start time)
   // 
   //  actual_EndTime        ACTUAL — Time at which the TRIGGER signal     DTL
   //                      went low (event end time)
   // 
   //  actual_Duration        ACTUAL — Event duration              LTime
   // 
   //  actual_DurationSec       ACTUAL — Event duration in seconds           REAL
   //  ――――――――――――――――――――――――――――――――――――――――――
   //  Block returned signals.
   // 
   // 
   // 
   // ▂▂▂▂▂▂▂▂▂▂▂▂▂▂▂▂▂▂▂▂▂▂▂▂▂▂▂▂▂▂▂▂▂▂▂▂▂▂▂▂▂▂▂▂
   // 3.1     Timing an event
   // 
   // 
   // The block constantly monitors the TRIGGER parameter; if a rising edge is seen on the TRIGGER 
   // parameter (point ① in the figure below), the Controller RTC is read and its value is stored in 
   // actual_StartTime, at the same time the running signal (status_Running) is activated.
   // 
   // The block continues to monitor the TRIGGER parameter, when a falling edge is detected 
   // (point ②), the RTC is read once more and its value is stored in actual_EndTime, and the running 
   // signal (status_Running) is deactivated.
   // 
   // Once the end time is stored, the following calculation is carried out:
   // 
   // 
   // ┌───────────────────────────┐
   // │ actual_Duration =  actual_EndTime ─ actual_StartTime    │
   // └───────────────────────────┘
   // 
   // 
   //                     ①            ②
   //   TRIGGER │             ┏━━━━━━━━━━━━┓
   //         │             ┃               ┃
   //         │             ┃               ┃
   //         │             ┃               ┃
   //         │             ┃               ┃                              
   //         ┼━━━━━━━━━━━━╶╶╶╶╶╶╶╶╶╶╶╶╶━━━━━━━━━━ time
   //                  ↗             ↖
   //            actual_StartTime ╎            ╎ actual_EndTime
   //    DTL#2020-04-18-09:34:25.899548353        DTL#2020-04-18-09:34:36.004744916
   // 
   //                    ╎               ╎                      actual_Duration
   //                                      LT#10S_105MS_196US_563NS
   //                    ╎               ╎  
   //                                                     actual_DurationSec
   //                    ╎               ╎                              10.10519
   // 
   //         │status_Running      ┏━━━━━━━━━━━━┓
   //         │             ┃               ┃
   //         │             ┃               ┃
   //         │             ┃               ┃
   //         │             ┃               ┃
   //         ┼━━━━━━━━━━━━╶╶╶╶╶╶╶╶╶╶╶╶╶━━━━━━━━━━
   // 
   // 
   // 
   // ▂▂▂▂▂▂▂▂▂▂▂▂▂▂▂▂▂▂▂▂▂▂▂▂▂▂▂▂▂▂▂▂▂▂▂▂▂▂▂▂▂▂▂▂
   // 3.1     Date and time data types
   // 
   // 
   // Both the start and end times (actual_StartTime and actual_EndTime) are of the type DTL 
   // (date time long), this itself is a data structure in the form:
   // 
   // 
   //  DTL Data Structure
   //  ――――――――――――――――――――――――――――――――――――――――――
   //  SIGNAL NAME          FUNCTION                     TYPE
   //  ――――――――――――――――――――――――――――――――――――――――――
   //  YEAR             Year (returns a value in the range 1970 to 2262)     UInt
   //  MONTH            Month (1-12 representing Jan to Dec)        USInt
   //  DAY              Day of month (1-31)                USInt
   //  WEEKDAY          Day of week (1-7, where 1=Sunday, 7=Saturday)    USInt
   //  HOUR           Hour of day (0-23)                   USInt
   //  MINUTE           Minutes (0-59)                   USInt
   //  SECOND            Seconds (0-59)                  USInt
   //  NANOSECOND        Nanoseconds (0-999,999,999)           UDint
   //  ――――――――――――――――――――――――――――――――――――――――――
   // 
   // 
   // When displayed, it has the format:
   // 
   //       DTL#2020-04-18-09:34:25.899548353
   // 
   //  I.e.      18th April 2020 at 09:43:25 AM and 899,548,353 ns.
   // 
   // The calculated duration (actual_Duration) is of data type LTime (long time).
   // 
   // The LTime data type is essentially an 8-byte number (64-bit number) that stores a time value in 
   // nanoseconds. In the above example, the actual_Duration has the formatted value of:
   // 
   //       LT#10S_105MS_196US_563NS
   // 
   //  I.e.      10 seconds, 105 milliseconds, 196 microseconds and 563 nanoseconds.
   // 
   // It is shown in this format, because TIA portal understands the LTime data type and is able to 
   // interpret the value as days, hours, minute, seconds, milliseconds, microseconds and 
   // nanoseconds. 
   // 
   // In practice, the actual_Duration simply (in this example) holds a very large number:
   // 
   //       10,105,196,563
   // 
   // This is the duration of the event in nanoseconds (i.e. 10,105,196,563 nanoseconds). To convert 
   // the number to seconds, simply divide by 1,000,000,000 (or 1 × 10^9); this would give:
   // 
   //       10.105196563 seconds
   // 
   // The reason the duration is specified as an LTime rather that DTL is that, somewhat confusingly, 
   // DTL is a relative measure of time (relative to 1st January, 1970), if the above duration were 
   // represented as a DTL value it would read:
   // 
   //       DTL#1970-01-01-00:00:10.105196563
   // 
   // Hours, minutes and seconds are OK, but the date part doesn’t make sense (to make it 
   // meaningful, 1970 must be subtracted from the YEAR value and 1 from both the MONTH and 
   // DAY values).
   // 
   // The LTime data type can store a duration of up to 106,751 days (about 300 years) and while not 
   // perfect, it seems long enough for most practical situations (possibly not for geological 
   // applications).
   // 
   // The actual_Duration in LTime format is very accurate, but it is an unwieldly data type, to provide a 
   // more user friendly (although less accurate) format, the actual_Duration signal is converted to a 
   // real number giving the duration in seconds, this is stored in the actual_DurationSec signal. In the 
   // above example: 
   // 
   //       actual_DurationSec has the value 10.10519 seconds
   // 
   // It is less accurate, it does not resolve to nanoseconds; however, it is easier to use and display 
   // and is accurate enough for most applications.
   // 
   // 
   // 
   // ▁▁▁▁▁▁▁▁▁▁▁▁▁▁▁▁▁▁▁▁▁▁▁▁▁▁▁▁▁▁▁▁▁▁▁▁▁▁▁▁▁▁▁▁
   // A note on real numbers
   // 
   // 
   // The LTime format is very accurate, it is basically counting nanoseconds, and because it is 64-bits 
   // long it can count up to very high values (about 584 years at nanosecond resolution).
   // 
   // Real numbers however, are limited to 32-bits and suffer from precision loss, this results from the 
   // fact that the real number has an accuracy of “about” 7 decimal digits, for example 20365.45, 
   // 20.43728, 1.482967, 0.3356428, &c. Essentially, the bigger the number, the fewer the decimal 
   // places — a total of 7 decimal digits.
   // 
   // Very big and very small numbers can be represented by adding trailing zeros for big numbers 
   // (e.g. 3275625000) and leading zeros for small numbers (0.000003275625) in both these 
   // examples, there are only 7 decimal digits, just shifted effectively left or right.
   // 
   // This type of representation is usually handled by applying scientific notation, the number 
   // 1,568,497,000,000 would be represented as 1.568497 × 10^12, it only has 7 decimal digits, 
   // the number 1,568,497,132,792, would be represented as exactly the same value, the 132,792 
   // part of the number cannot be resolved and are lost.
   // 
   //                ━━━   ⬙⬙⬙⬙⬙⬙   ━━━
END_REGION

REGION Network 4: Example — Block description — Sections 4 to 11
   // ▄▄▄▄▄▄▄▄▄▄▄▄▄▄▄▄▄▄▄▄▄▄▄▄▄▄▄▄▄▄▄▄▄▄▄▄▄▄▄▄▄▄▄▄
   // 4.     PARAMETERS
   // 
   // 
   // The following parameters are associated with the block:
   // 
   //  
   //  ――――――――――――――――――――――――――――――――――――――――――
   //  PARAM         FUNCTION                    TYPE      IN-OUT 
   //  ――――――――――――――――――――――――――――――――――――――――――
   //  SYS_SIGNALS      Common system signals              UT21000    In
   //           logic and timing signals for parametric access
   // 
   //  TRIGGER       Event trigger signal (a rising edge marks the     Bool   In
   //           start of the event, the falling edge the end)
   // 
   //  STATIC_DATA     Data structure that holds the configuration data     UT02001    In
   // 
   //  DYNAMIC_DATA      Stores the results of the event timing       UT38151    InOut
   //  ――――――――――――――――――――――――――――――――――――――――――
   // 
   // 
   //                ━━━   ⬙⬙⬙⬙⬙⬙   ━━━
   // 
   // 
   // 
   // ▄▄▄▄▄▄▄▄▄▄▄▄▄▄▄▄▄▄▄▄▄▄▄▄▄▄▄▄▄▄▄▄▄▄▄▄▄▄▄▄▄▄▄▄
   // 5.     DATA STRUCTURES AND USAGE (AND INSTANCE DATA BLOCKS)
   // 
   // 
   // The block has the following associated data structure:
   // 
   // 
   //  ――――――――――――――――――――――――――――――――――――――――――
   //  DATA STRUCTURE             DESCRIPTION
   //  ――――――――――――――――――――――――――――――――――――――――――
   //  UT01000_St_SysRevision          Revision information for this block    See FC01001
   //  UT01001_St_SysLicence           Licence information for this block  See FC01001
   //  UT21000_Dy_SysSignals           System signals for logic and timing  See FC01001
   //  UT38151_Dy_SubTimeEventRTC        Dynamic data structure for the event timing block
   //  ――――――――――――――――――――――――――――――――――――――――――
   // 
   // 
   // 
   // ▂▂▂▂▂▂▂▂▂▂▂▂▂▂▂▂▂▂▂▂▂▂▂▂▂▂▂▂▂▂▂▂▂▂▂▂▂▂▂▂▂▂▂▂
   // 5.1     UT38151_Dy_TimeEventRTC
   // 
   // 
   // Stores the timing values for the event:
   // 
   // 
   //  UT38151_Dy_TimeEventRTC
   //  ――――――――――――――――――――――――――――――――――――――――――
   //  SIGNAL NAME          FUNCTION                     TYPE
   //  ――――――――――――――――――――――――――――――――――――――――――
   //  status_Running      STATUS — The event timer is running         Bool
   // 
   //  actual_StartTime      ACTUAL — Time at which the TRIGGER signal        DTL
   //                      went high (event start time)
   // 
   //  actual_EndTime        ACTUAL — Time at which the TRIGGER signal     DTL
   //                      went low (event end time)
   // 
   //  actual_Duration        ACTUAL — Event duration              LTime
   // 
   //  actual_DurationSec       ACTUAL — Event duration in seconds           REAL
   //  ――――――――――――――――――――――――――――――――――――――――――
   // 
   // 
   //                ━━━   ⬙⬙⬙⬙⬙⬙   ━━━
   // 
   // 
   // 
   // ▄▄▄▄▄▄▄▄▄▄▄▄▄▄▄▄▄▄▄▄▄▄▄▄▄▄▄▄▄▄▄▄▄▄▄▄▄▄▄▄▄▄▄▄
   // 6.     CONSTANTS AND TEMPORARY (LOCAL) DATA
   // 
   // 
   // The following constants and temporary data storage are used:
   // 
   // 
   //  Temporary (local) data
   //  ――――――――――――――――――――――――――――――――――――――――――
   //  SIGNAL NAME          FUNCTION                  TYPE
   //  ――――――――――――――――――――――――――――――――――――――――――
   //  revInfo             Revision information for the block         UT01000
   //  licInfo           Licensing information for the block      UT01001
   //  wrkInt           Working storage area (integer)          Int
   //  wrkReal           Working storage (Real)             Real
   //  wrkLInt            Working storage area (long integer)        LInt
   //  ――――――――――――――――――――――――――――――――――――――――――
   // 
   // 
   //                ━━━   ⬙⬙⬙⬙⬙⬙   ━━━
   // 
   // 
   // 
   // ▄▄▄▄▄▄▄▄▄▄▄▄▄▄▄▄▄▄▄▄▄▄▄▄▄▄▄▄▄▄▄▄▄▄▄▄▄▄▄▄▄▄▄▄
   // 7.     BLOCK CALLS
   // 
   // 
   // There are no PAL block calls from within this block.
   // 
   //                ━━━   ⬙⬙⬙⬙⬙⬙   ━━━
   // 
   // 
   // 
   // ▄▄▄▄▄▄▄▄▄▄▄▄▄▄▄▄▄▄▄▄▄▄▄▄▄▄▄▄▄▄▄▄▄▄▄▄▄▄▄▄▄▄▄▄
   // 8.     ASSOCIATED BLOCKS
   // 
   // 
   // This is a stand-alone block and is not associated with any other blocks.
   // 
   //                ━━━   ⬙⬙⬙⬙⬙⬙   ━━━
   // 
   // 
   // 
   // ▄▄▄▄▄▄▄▄▄▄▄▄▄▄▄▄▄▄▄▄▄▄▄▄▄▄▄▄▄▄▄▄▄▄▄▄▄▄▄▄▄▄▄▄
   // 9.     SYSTEM BLOCK CALLS AND SYSTEM DATA TYPES
   // 
   // 
   // The following calls are made to system blocks:
   // 
   // 
   //  System block calls
   //  ――――――――――――――――――――――――――――――――――――――――――
   //  BLOCK          TITLE             DESCRIPTION  
   //  ――――――――――――――――――――――――――――――――――――――――――
   //  RD_LOC_T             Read the local RTC time    Reads the CPU real time clock 
   //  ――――――――――――――――――――――――――――――――――――――――――
   // 
   // 
   // There are no special system data types used.
   // 
   //                ━━━   ⬙⬙⬙⬙⬙⬙   ━━━
   // 
   // 
   // 
   // ▄▄▄▄▄▄▄▄▄▄▄▄▄▄▄▄▄▄▄▄▄▄▄▄▄▄▄▄▄▄▄▄▄▄▄▄▄▄▄▄▄▄▄▄
   // 10.     SPECIAL PROPERTIES AND REQUIREMENTS
   // 
   // 
   // 
   // ▂▂▂▂▂▂▂▂▂▂▂▂▂▂▂▂▂▂▂▂▂▂▂▂▂▂▂▂▂▂▂▂▂▂▂▂▂▂▂▂▂▂▂▂
   // 10.1   Block optimisation
   // 
   // 
   // Block optimisation is ACTIVE for this block
   // 
   // 
   // 
   // ▂▂▂▂▂▂▂▂▂▂▂▂▂▂▂▂▂▂▂▂▂▂▂▂▂▂▂▂▂▂▂▂▂▂▂▂▂▂▂▂▂▂▂▂
   // 10.2   Calling requirements
   // 
   // 
   // There are no special calling requirements for this block.
   // 
   // 
   // 
   // ▂▂▂▂▂▂▂▂▂▂▂▂▂▂▂▂▂▂▂▂▂▂▂▂▂▂▂▂▂▂▂▂▂▂▂▂▂▂▂▂▂▂▂▂
   // 10.3   Other properties
   // 
   // 
   // This block does not require the usual SYS_SIGNALS logic and timing data.
   // 
   //                ━━━   ⬙⬙⬙⬙⬙⬙   ━━━
   // 
   // 
   // 
   // ▄▄▄▄▄▄▄▄▄▄▄▄▄▄▄▄▄▄▄▄▄▄▄▄▄▄▄▄▄▄▄▄▄▄▄▄▄▄▄▄▄▄▄▄
   // 11.     EXAMPLE USAGE
   // 
   // 
   // The following shows a typical deployment of FC18151:
   // 
   //                      ┌─────────────
   //        ──────────────┤ FC18151
   //                      ├───────────
   //                 %M100.0    │
   //               "Event001"   ─┤ TRIGGER
   //                      │
   //     "DB38151_Dy_TimeEventRTC".Event001 ─┤ DYNAMIC_DATA
   //                      │
   //                      │             │
   //                                    │
   //                           ─────────┘
   // 
   //               ━━━   ⬙⬙⬙⬙⬙⬙   ━━━
   // 
   // 
   // ██████████████ █ █ █ █  END   █ █ █ █ ██████████████
END_REGION

REGION Network 5: Example — Current revision and modification history
   // ▄▄▄▄▄▄▄▄▄▄▄▄▄▄▄▄▄▄▄▄▄▄▄▄▄▄▄▄▄▄▄▄▄▄▄▄▄▄▄▄▄▄▄▄
   // MODIFICATION HISTORY
   // 
   // 
   // The revision data shown here, in the network comments, contains additional information 
   // reflecting the software development workflow under the version control system (VCS) employed 
   // to track all software changes.
   // 
   // The VCS in use is the Git Source Code Management system in conjunction with the GitHub online 
   // hosting system. The software in its entirety is available in the GitHub remote repository:
   // 
   //      https://github.com/practicalseries/PS2001-pal-software
   // 
   // The repository is public and can be freely copied (forked in GitHub terminology) and used 
   // under the MIT licence. 
   // 
   // The MIT licence is reproduced in full in the last network of this software module.
   // 
   // 
   //  ―――――――――――――――――――――――――――――――――――――――――――
   //  DATE       REVISION             MASTER BRANCH     DEV
   //          (nnn.amm)   COMMIT TAG    (Base ---> Merge)    BRANCH   Author
   //  ———————————————————————————————————————————
   //  2020.11.09    001.000   D0003      D0002 D0003  None    M. Gledhill
   //                        FC01001 — RELEASED FOR USE
   //                          Merge back to master branch
   //  
   //  2020.11.09    001.000   D0002A-001.000   D0002 N/A     D0002A   M. Gledhill
   //                        FC01001 — Post test released for use
   // 
   //  2020.11.08    000.801   D0002A-000.801   D0002 N/A     D0002A   M. Gledhill
   //                        FC01001 — Released for SMT
   // 
   //  2020.11.04    000.102   D0002A-000.102   D0002 N/A     D0002A   M. Gledhill
   //                        FC01001 — Incremental build
   // 
   //  2020.11.03    000.101   D0002A-000.101   D0002 N/A     D0002A   M. Gledhill
   //                        FC01001 — Block created
   //  ———————————————————————————————————————————
   //   Where: nnn  =  Major revision
   //         a  =  Type (1-7 Development, 8 Proving, 9 Qualification, 0 Release)
   //       mm  =  Minor revision (must be 00 if a = 0)
   //         Block properties version number should be set to nn.a (only one decimal place)
   // 
   // ▄▄▄▄▄▄▄▄▄▄▄▄▄▄▄▄▄▄▄▄▄▄▄▄▄▄▄▄▄▄▄▄▄▄▄▄▄▄▄▄▄▄▄▄
   RUNG wire#powerrail
      I_Contact( #SYS_SIGNALS._False )
      wire#w1
      S_Move(in := 'FC01001', out => #revInfo.REV_BLOCK)
   END_RUNG
   RUNG wire#w1
      S_Move(in := '001.000', out => #revInfo.REV_NUMBER)
   END_RUNG
   RUNG wire#w1
      S_Move(in := '2020.11.09', out => #revInfo.REV_DATE)
   END_RUNG
   RUNG wire#w1
      S_Move(in := 'M. Gledhill', out => #revInfo.REV_AUTHOR)
   END_RUNG
   // the same network as SCL:
   IF NOT #SYS_SIGNALS._False THEN
       #revInfo.REV_BLOCK := 'FC01001';
       #revInfo.REV_NUMBER := '001.000';
       #revInfo.REV_DATE := '2020.11.09';
       #revInfo.REV_AUTHOR := 'M. Gledhill';
   END_IF;
END_REGION

REGION Network 6: Example — Headings, lists and indented text
   // ▀▀▀▀▀▀▀▀▀▀▀▀▀▀▀▀▀▀▀▀▀▀▀▀▀▀▀▀▀▀▀▀▀▀▀▀▀▀▀▀▀▀▀▀
   // ↳
   // TITLE:    HEADINGS, LISTS AND INDENTED TEXT
   // ↳
   // ▄▄▄▄▄▄▄▄▄▄▄▄▄▄▄▄▄▄▄▄▄▄▄▄▄▄▄▄▄▄▄▄▄▄▄▄▄▄▄▄▄▄▄▄[3 empty lines below]
   // ↳
   // ↳
   // ↳
   // Lorem ipsum dolor sit amet, consectetur adipiscing elit, sed do eiusmod tempor incididunt ut 
   // labore et dolore magna aliqua. Euismod lacinia at quis risus sed. Semper feugiat nibh sed 
   // pulvinar proin gravida hendrerit.
   // ↳
   //                ━━━   ⬙⬙⬙⬙⬙⬙   ━━━[1 empty line above]
   // ↳
   // ↳
   // ↳
   // ▄▄▄▄▄▄▄▄▄▄▄▄▄▄▄▄▄▄▄▄▄▄▄▄▄▄▄▄▄▄▄▄▄▄▄▄▄▄▄▄▄▄▄▄[3 empty lines above, 2 after title]
   // 1.     [MAIN SECTION — ALL UPPERCASE — IF UNNUMBERED STARTS AT LEFT EDGE]
   // 10.     [MAIN SECTION — ALL UPPERCASE — IF UNNUMBERED STARTS AT LEFT EDGE]
   // ↳
   // ↳
   // Lorem ipsum dolor sit amet, consectetur adipiscing elit, sed do eiusmod tempor incididunt ut 
   // labore et dolore magna aliqua. Euismod lacinia at quis risus sed. Semper feugiat nibh sed 
   // pulvinar proin gravida hendrerit.
   // ↳
   //                ━━━   ⬙⬙⬙⬙⬙⬙   ━━━[1 empty line above]
   // ↳
   // ↳
   // ↳
   // ▂▂▂▂▂▂▂▂▂▂▂▂▂▂▂▂▂▂▂▂▂▂▂▂▂▂▂▂▂▂▂▂▂▂▂▂▂▂▂▂▂▂▂▂[3 empty lines above, 2 after title]
   // 1.1     [Subsection, two single digits   — Sentence case — if unnumbered, starts at left edge]
   // 10.1   [Subsection, one double digit   — Sentence case — if unnumbered, starts at left edge]
   // 10.10    [Subsection, two double digits — Sentence case — if unnumbered, starts at left edge]
   // ↳
   // ↳
   // Lorem ipsum dolor sit amet, consectetur adipiscing elit, sed do eiusmod tempor incididunt ut 
   // labore et dolore magna aliqua. Euismod lacinia at quis risus sed. Semper feugiat nibh sed 
   // pulvinar proin gravida hendrerit.
   // ↳
   //                ━━━   ⬙⬙⬙⬙⬙⬙   ━━━[1 empty line above]
   // ↳
   // ↳
   // ↳
   // ▁▁▁▁▁▁▁▁▁▁▁▁▁▁▁▁▁▁▁▁▁▁▁▁▁▁▁▁▁▁▁▁▁▁▁▁▁▁▁▁▁▁▁▁[3 empty lines above, 2 after title]
   // 1.1.1     [Inline, three single digits   — Sentence case — if unnumbered, starts at left edge]
   // 10.1.1   [Inline, one double digit   — Sentence case — if unnumbered, starts at left edge]
   // 10.10.1   [Inline, two double digits    — Sentence case — if unnumbered, starts at left edge]
   // 10.10.10 [Inline, three double digits — Sentence case — if unnumbered, starts at left edge]
   // ↳
   // ↳
   //    •   [Lists — non-numbered]
   //    ① [Lists — numbered]
   //    1.  [Lists — numbered single digit   — less than 10 entries]
   //      1.  [Lists — numbered single digit   — 10 or more entries]
   //    10.  [Lists — numbered double digit — 10 or more entries]
   // 
   //    1.  Communication handling
   //      Executes system to system communications (Controller to Controller, point-to-point,
   //      ProfiBus FMS &c.)
   //    2.  Subroutine functions
   //      Various subroutines (called by other block) to execute particular functions 
   //      (subroutines are organised into similar function areas)
   //    3.  Normal (non-error) interrupt functions
   //      Usually associated with specific OBs, interrupts generated by standard system events
   //      (time of day, cyclic, hardware &c.)
   // 
   // Note:    Bipolar and unipolar instruments have different tolerances, a 0-20 mA unipolar signal
   //      has a full instrument range of 16 mA and the 2.5% tolerance will thus be ±0.4 mA 
   // 
   // ――――――――――
   // ¹         Footnotes can use the characters ¹, ² and ³ to indicate the footnote number
   //      Second lines are identical to those for notes.
   // ――――――――――
   // ↳
   //                ━━━   ⬙⬙⬙⬙⬙⬙   ━━━
   // ↳
   // ↳
   // ██████████████ █ █ █ █  END   █ █ █ █ ██████████████
   // ↳
END_REGION

REGION Network 7: Example — Body text
   // ▀▀▀▀▀▀▀▀▀▀▀▀▀▀▀▀▀▀▀▀▀▀▀▀▀▀▀▀▀▀▀▀▀▀▀▀▀▀▀▀▀▀▀▀
   // 
   // TITLE:    BODY TEXT (AN EXAMPLE)
   // 
   // ▄▄▄▄▄▄▄▄▄▄▄▄▄▄▄▄▄▄▄▄▄▄▄▄▄▄▄▄▄▄▄▄▄▄▄▄▄▄▄▄▄▄▄▄
   // 
   // 
   // Normal (body) text is left justified to the left hand edge of the comment area; manual line-breaks
   // must be inserted when the text exceeds the range of the title bars (lines at the top of this block
   // and above each section and subsection — exactly 44 em-spaces).
   // 
   // The following fragment highlights this: 
   // 
   // The alignments in Figure 7.4 are such that the leading edge (left side) of any indented character
   // is aligned with the leading edge of an em-space in a line of em-spaces that span the page (this
   // can be seen with the chequered patterns in the screen shot — all indents line up with the left
   // edge of an em-space).
   // 
   // The problem with this is that the alphanumeric characters are not all the same width and
   // generally, they are not one em-space wide (there are no characters that are one em wide, not
   // even the M, which is odd given that that is how the em unit was derived, see here).
   // With the TIA Portal font, one em is exactly the same width as four normal space characters (a 
   // normal space being the character entered when the space bar is pressed). The alphanumeric 
   // characters (and in fact, all the characters) in the TIA Portal font have the peculiarity that they are
   // all a multiple of ⅓ of a normal space , the “i" for example is one normal space wide, “a” is 2⅓
   // normal space characters wide and “m” is 2⅔ normal space characters wide.
   // 
   // This “feature?” of the font is a distinct advantage; it means that is possible to always bring things
   // back into true alignment by using the range of whitespace characters. There are five such 
   // whitespace characters.
   // 
   // The width of the page is approximately 3.38 lowercase alphabets:
   // 
   // abcdefghijklmnopqrstuvwxyzabcdefghijklmnopqrstuvwxyzabcdefghijklmnopqrstuvwxyzabcdefghij
   // 
   // This averages at about 78 (non-space) characters per line.
   // 
   // A comment field can contain 65000 characters (approx.) including spaces and line breaks.
   // 
   // This broadly equates to 670 lines of standard text, approximately 13000 words.
   // ↳
   //                ━━━   ⬙⬙⬙⬙⬙⬙   ━━━
   // ↳
   // ↳
   // ██████████████ █ █ █ █  END   █ █ █ █ ██████████████
   // ↳
END_REGION

REGION Network 8: Example — Standard Tables
   // ▀▀▀▀▀▀▀▀▀▀▀▀▀▀▀▀▀▀▀▀▀▀▀▀▀▀▀▀▀▀▀▀▀▀▀▀▀▀▀▀▀▀▀▀
   // 
   // TITLE:    STANDARD TABLES (EXAMPLES)
   // 
   // ▄▄▄▄▄▄▄▄▄▄▄▄▄▄▄▄▄▄▄▄▄▄▄▄▄▄▄▄▄▄▄▄▄▄▄▄▄▄▄▄▄▄▄▄
   // 
   // 
   // 
   // Tables always have 2 blank lines above and 2 blank lines below.
   // 
   // ▌▌▌▌▌▌▌▌▌▌▌▌▌▌▌▌▌▌PARAMETER TABLE▐▐▐▐▐▐▐▐▐▐▐▐▐▐▐▐▐▐
   // ↳
   // ↳
   //  ――――――――――――――――――――――――――――――――――――――――――
   //  PARAM         FUNCTION                    TYPE      IN-OUT 
   //  ――――――――――――――――――――――――――――――――――――――――――
   //  SYS_SIGNALS      The system logic and timing signals for       UT21000    In
   //           parametric access
   // 
   //  RAW_ANALOG      The unscaled analogue input (input word         Word     In
   //           address for the IO card to which the instrument 
   //           is connected)
   // 
   //  RAW_MIN     Minimum value of the analogue input range      Int      In
   //           (see Table 3.1 to Table 3.3 for typical values)
   // 
   //  RAW_MAX       Maximum value of the analogue input range      Int      In
   //           (see Table 3.1 to Table 3.3 for typical values)
   // 
   //  SCALE_MIN    Calibrated lower value of the instrument       Real      In
   //           range in engineering units
   // 
   //  SCALE_MAX      Calibrated upper value of the instrument      Real      In
   //           range in engineering units
   // 
   //  STATIC_DATA     The static data associated with the PID loop       UT10001 In
   // 
   //  DYNAMIC_DATA      Stores the results of the event timing       UT38151    InOut
   //  ――――――――――――――――――――――――――――――――――――――――――
   // ↳
   // ↳
   // 
   // ▌▌▌▌▌▌▌▌▌▌▌▌▌▌▌▌▌ DATA STRUCTURE LIST ▐▐▐▐▐▐▐▐▐▐▐▐▐▐▐▐▐
   // ↳
   // ↳
   //  ――――――――――――――――――――――――――――――――――――――――――
   //  DATA STRUCTURE             DESCRIPTION
   //  ――――――――――――――――――――――――――――――――――――――――――
   //  UT01000_St_SysRevision          Revision information for this block    See FC01000
   //  UT01001_St_SysLicence           Licence information for this block  See FC01000
   //  UT21000_Dy_SysSignals           System signals for logic and timing  See FC01000
   // 
   //  UT02001_St_InstAnalogRead      Static data structure for an analogue instrument.
   //                     Holds configuration information, instrument ranges 
   //                     and scaling, alarm/warning thresholds &c.
   // 
   //  UT22001_Dy_InstAnalogRead        Dynamic data structure for an analogue instrument.
   //                     Current scaled instrument reading, alarm status, 
   //                     operating modes, timer values &c.
   //  ――――――――――――――――――――――――――――――――――――――――――
   // ↳
   // ↳
   // 
   // ▌▌▌▌▌▌▌▌▌▌   DATA STRUCTURE CONTENTS AND INSTANCE DBs   ▐▐▐▐▐▐▐▐▐▐
   // ↳
   // ↳
   //  UT38151_Dy_TimeEventRTC
   //  ――――――――――――――――――――――――――――――――――――――――――
   //  SIGNAL NAME          FUNCTION                     TYPE
   //  ――――――――――――――――――――――――――――――――――――――――――
   //  status_Running      STATUS — The event timer is running         Bool
   // 
   //  actual_StartTime      ACTUAL — Time at which the TRIGGER signal        DTL
   //                      went high (event start time)
   // 
   //  actual_EndTime        ACTUAL — Time at which the TRIGGER signal     DTL
   //                      went low (event end time)
   // 
   //  actual_Duration        ACTUAL — Event duration              LTime
   // 
   //  actual_DurationSec       ACTUAL — Event duration in seconds           REAL
   //  ――――――――――――――――――――――――――――――――――――――――――
   // ↳
   // ↳
   // 
   // ▌▌▌▌▌▌▌▌▌▌▌▌▌▌▌  CONSTANTS AND LOCAL DATA  ▐▐▐▐▐▐▐▐▐▐▐▐▐▐▐
   // 
   // [Keep local and constant data function description to one line and no gaps between rows]
   // ↳
   // ↳
   //  CONSTANTS DATA
   //  ――――――――――――――――――――――――――――――――――――――――――
   //  SIGNAL NAME       Value    FUNCTION                  TYPE
   //  ――――――――――――――――――――――――――――――――――――――――――
   //  k_TIME_OP_MIN      0.21      Minimum value for the operation timer     Real
   //  ――――――――――――――――――――――――――――――――――――――――――
   // ↳
   // ↳
   //  TEMPORARY (LOCAL) DATA
   //  ――――――――――――――――――――――――――――――――――――――――――
   //  SIGNAL NAME          FUNCTION                     TYPE
   //  ――――――――――――――――――――――――――――――――――――――――――
   //  wrkPercentPV          Process Variable as a percentage of inst. range     Real
   //  wrkPercentSP          Setpoint as a percentage of PV instrument range     Real
   //  wrkPercentDB         Deadband as a percentage of PV instrument range    Real
   //  wrkGain          Gain (adjusted for reverse/normal Acting)      Real
   //  wrkCycTime          Cyclic execution time (TIME format)         Time
   //  ――――――――――――――――――――――――――――――――――――――――――
   // ↳
   // ↳
   // 
   // ▌▌▌▌▌▌▌▌▌▌▌▌▌▌▌▌▌▌▌  BLOCK LIST  ▐▐▐▐▐▐▐▐▐▐▐▐▐▐▐▐▐▐▐
   // ↳
   // ↳
   //  BLOCK CALLS
   //  ――――――――――――――――――――――――――――――――――――――――――
   //  BLOCK          TITLE             DESCRIPTION  
   //  ――――――――――――――――――――――――――――――――――――――――――
   //  FC18001         StdSubScaleAI        Scales an analogue input signal 
   //                            Continuation line
   //  ――――――――――――――――――――――――――――――――――――――――――
   // ↳
   // ↳
   //  ASSOCIATED BLOCKS
   //  ――――――――――――――――――――――――――――――――――――――――――
   //  BLOCK          TITLE             DESCRIPTION  
   //  ――――――――――――――――――――――――――――――――――――――――――
   //  FC17102         StdCommsWrite65K       Write data partner block
   //                            Continuation line 
   //  ――――――――――――――――――――――――――――――――――――――――――
   // ↳
   // ↳
   // 
   // ▌▌▌▌▌▌▌▌▌▌▌▌▌▌▌▌▌  SYSTEM BLOCK LIST   ▐▐▐▐▐▐▐▐▐▐▐▐▐▐▐▐▐
   // ↳
   // ↳
   //  SYSTEM BLOCK CALLS
   //  ――――――――――――――――――――――――――――――――――――――――――
   //  BLOCK          TITLE             DESCRIPTION  
   //  ――――――――――――――――――――――――――――――――――――――――――
   //  RD_LOC_T             Read the local RTC time    Reads the CPU real time clock 
   //  (FC804)                        Continuation line 
   //                            Continuation line
   //  ――――――――――――――――――――――――――――――――――――――――――
   // ↳
   // ↳
   // 
   // ▌▌▌▌▌▌▌▌▌▌▌▌▌▌▌▌▌▌▌▌▌▌▐▐▐▐▐▐▐▐▐▐▐▐▐▐▐▐▐▐▐▐▐▐
   // ↳
   //                ━━━   ⬙⬙⬙⬙⬙⬙   ━━━
   // ↳
   // ↳
   // ██████████████ █ █ █ █  END   █ █ █ █ ██████████████
   // ↳
END_REGION

REGION Network 9: Example — Other tables
   // ▀▀▀▀▀▀▀▀▀▀▀▀▀▀▀▀▀▀▀▀▀▀▀▀▀▀▀▀▀▀▀▀▀▀▀▀▀▀▀▀▀▀▀▀
   // 
   // TITLE:    OTHER TABLES (EXAMPLES)
   // 
   // ▄▄▄▄▄▄▄▄▄▄▄▄▄▄▄▄▄▄▄▄▄▄▄▄▄▄▄▄▄▄▄▄▄▄▄▄▄▄▄▄▄▄▄▄
   // 
   // 
   // 
   // Tables always have 2 blank lines above and 2 blank lines below.
   // 
   // 
   // ▌▌▌▌▌▌▌▌▌▌▌▌▌▌▌▌▌  TWO COLUMN TABLE ▐▐▐▐▐▐▐▐▐▐▐▐▐▐▐▐▐
   // ↳
   // ↳
   //  ――――――――――――――――――――――――――――――――――――――――――
   //  IO TYPE            DESCRIPTION
   //  ――――――――――――――――――――――――――――――――――――――――――
   //  ET200MP         Standard IO high density IO for the S7-1500 range
   // 
   //  ET200M           Standard IO high density IO for the S7-300 range, 
   //               can be used as remote IO for the S7-1500
   //  ――――――――――――――――――――――――――――――――――――――――――
   // ↳
   // ↳
   // 
   // ▌▌▌▌▌▌▌▌▌▌▌▌▌▌▌▌▌THREE COLUMN TABLE ▐▐▐▐▐▐▐▐▐▐▐▐▐▐▐▐▐
   // 
   // [Numerical table with number alignment to the right]
   // ↳
   // ↳
   //  ――――――――――――――――――――――――――――――――――――――――――
   //  PRESSURE           RAW SIGNAL           SCALED VAL
   //  ――――――――――――――――――――――――――――――――――――――――――
   //  -250.0 Pa                   0             -250.0 Pa
   //        0.0 Pa                  13824            0.0 Pa
   //   250.0 Pa                  27648              250.0 Pa
   //  ――――――――――――――――――――――――――――――――――――――――――
   // ↳
   // ↳
   // 
   // ▌▌▌▌▌▌▌▌▌▌▌▌▌▌▌▌▌ FOUR COLUMN TABLE ▐▐▐▐▐▐▐▐▐▐▐▐▐▐▐▐▐
   // 
   // [Numerical table with number alignment to the right]
   // ↳
   // ↳
   //  ――――――――――――――――――――――――――――――――――――――――――
   //  RAW MIN       RAW MAX      SCALED MIN       SCALED MAX
   //  ――――――――――――――――――――――――――――――――――――――――――
   //        0        27648        -250.0 Pa        250.0 Pa
   //  ――――――――――――――――――――――――――――――――――――――――――
   // ↳
   // ↳
   // 
   // ▌▌▌▌▌▌▌▌▌▌▌▌▌▌▌▌▌  TABLE WITH HEADING  ▐▐▐▐▐▐▐▐▐▐▐▐▐▐▐▐▐
   // 
   // [Numerical table with number alignment to the right]
   // ↳
   // ↳
   //  CURRENT SIGNALS
   //  ――――――――――――――――――――――――――――――――――――――――――
   //  SIGNAL TYPE     SIG MIN VAL      RAW_MIN     SIG MAX VAL     RAW_MAX
   //  ――――――――――――――――――――――――――――――――――――――――――
   //    4-20 mA      4 mA          0          20 mA       27648
   //    0-20 mA      0 mA          0          20 mA       27648
   //  -20 to 20 mA      -20 mA      -27648          20 mA       27648
   //  ――――――――――――――――――――――――――――――――――――――――――
   // ↳
   // ↳
   // 
   // ▌▌▌▌▌▌▌▌▌▌▌▌▌▌▌▌▌▌▌▌▌▌▐▐▐▐▐▐▐▐▐▐▐▐▐▐▐▐▐▐▐▐▐▐
   // ↳
   //                ━━━   ⬙⬙⬙⬙⬙⬙   ━━━
   // ↳
   // ↳
   // ██████████████ █ █ █ █  END   █ █ █ █ ██████████████
   // ↳
END_REGION

REGION Network 10: Example — Equations
   // ▀▀▀▀▀▀▀▀▀▀▀▀▀▀▀▀▀▀▀▀▀▀▀▀▀▀▀▀▀▀▀▀▀▀▀▀▀▀▀▀▀▀▀▀
   // 
   // TITLE:    EQUATIONS (EXAMPLES)
   // 
   // ▄▄▄▄▄▄▄▄▄▄▄▄▄▄▄▄▄▄▄▄▄▄▄▄▄▄▄▄▄▄▄▄▄▄▄▄▄▄▄▄▄▄▄▄
   // 
   // 
   // 
   // ┌─────────────────────────────────────┐
   // │                                                                                                              100                         │
   // │ SigPercent = (Signal ─ PV_RANGE_MIN) ╳ ---------------------------------------------------------------    │
   // │                    (PV_RANGE_MAX ─ PV_RANGE_MIN)    │
   // └─────────────────────────────────────┘
   // 
   // 
   // ┌───────────────────────┐
   // │        2.5               │
   // │ CalcValOOR = ------------ ╳ (RAW_MAX ─ RAW_MIN)   │
   // │       100               │
   // └───────────────────────┘
   // 
   // Mathematical operators:
   //    Large:  ┼ ─ ╳
   //    Small: + − × ÷ ± ≤ ≥
   // ↳
   //                ━━━   ⬙⬙⬙⬙⬙⬙   ━━━
   // ↳
   // ↳
   // ██████████████ █ █ █ █  END   █ █ █ █ ██████████████
   // ↳
END_REGION

REGION Network 11: Example — Figures
   // ▀▀▀▀▀▀▀▀▀▀▀▀▀▀▀▀▀▀▀▀▀▀▀▀▀▀▀▀▀▀▀▀▀▀▀▀▀▀▀▀▀▀▀▀
   // 
   // TITLE:    FIGURES (EXAMPLES)
   // 
   // ▄▄▄▄▄▄▄▄▄▄▄▄▄▄▄▄▄▄▄▄▄▄▄▄▄▄▄▄▄▄▄▄▄▄▄▄▄▄▄▄▄▄▄▄
   // 
   // 
   // 
   // Some example figures, always pad gaps with an EM-SPACE, where text is used add normal 
   // spaces with either a THREE-PER-EM space or a SIX-PER-EM space — one of these will give an
   // exact alignment.
   // 
   // These figures are included to show what is possible.
   // 
   // 
   // Figures have 1 blank line above and 1 below.
   // 
   //   → ┌────────┐
   // ┌───┤   IDLE   │
   // │   └───┬────┘
   // │       ↓
   // │       START
   // │       │
   // │   ┌───┴────┐ →
   // │   │  STARTING     ├───┐
   // │   └───┬────┘   │
   // │       ↓        │
   // │         Run*       ├────────────────────┐
   // │       │        │                    │
   // │   ┌───┴────┐ → │                    │
   // │   │        ├───┴───  Hold  ───┐          │
   // │   │        │             ↓          ↓
   // │   │        │         ┌───┴────┐ ┌───┴────┐
   // │   │        │         │  HOLDING    │ │ ErrHOLDING   │
   // │   │        │         └───┬────┘ └───┬────┘
   // │   │        │             Held*        ErrHeld*
   // │   │        │         ┌───┴────┐ ┌───┴────┐
   // │   │        │         │   HELD    │ │  ErrHELD   │
   // │   │  RUNNING     │         └───┬────┘ └───┬────┘
   // │   │        │              Resume         ErrResume
   // │   │        │         ┌───┴────┐ ┌───┴────┐
   // │  ┌┤        │         │   RESUMING    │ │  ErrRESUMING   │ 
   // │  ││        │         └───┬────┘ └───┬────┘  
   // │  ││        │             │          │
   // │  ││        │ ←           ↓          ↓
   // │  ││        │─────────────┴──────────┘
   // │  │└───┬────┘   Returns to previous step (running or starting)
   // │  ↓    ↓
   // │  │    │
   // │ Complete Complete*     Note: *indicates that the command is issued
   // │  │    │           automatically by the sequence (it
   // │  │┌───┴────┐      can also be triggered manually):
   // │  └┤ COMPLETING  │          1. Run
   // │   └───┬────┘          2. Complete
   // │       ↓               3. Completed
   // ↑     Completed*              4. Held
   // │       │               5. ErrHeld
   // │   ┌───┴────┐          6. Stopped
   // │   │  COMPLETED   │          7. Aborted
   // │   └───┬────┘
   // │       │
   // │              RetIdle*
   // │   ←   ↓
   // ├───────┘
   // │   
   // │
   // │     ABORT ROUTE                  STOPPING ROUTE
   // │Can be triggered in all states except       Can be triggered in all states except
   // │ IDLE, COMPLETED, ABORTING or            IDLE, COMPLETED, ABORTING, 
   // │       ABORTED                 ABORTED, STOPPING or STOPPED
   // │       │                       │
   // │       ↓                       ↓
   // │                Abort                                                                                       Stop
   // │       │                       │
   // │   ┌───┴────┐              ┌───┴────┐
   // ↑   │ ABORTING    │              │  STOPPING    │
   // │   └───┬────┘              └───┬────┘
   // │       ↓                       ↓
   // │              Aborted*                                                                                Stopped*
   // │       │                       │
   // │   ┌───┴────┐              ┌───┴────┐
   // │   │ ABORTED      │              │ STOPPED   │
   // │   └───┬────┘              └───┬────┘
   // │       │                       │
   // │      RetIdle (*)                                                                               RetIdle (*)
   // │  ←    ↓                       ↓
   // └───────┴───────────────────────┘
   // 
   // 
   // 
   // ▌▌▌▌▌▌▌▌▌▌▌▌▌▌▌▌▌▌   INLINE FIGURES ▐▐▐▐▐▐▐▐▐▐▐▐▐▐▐▐▐▐
   // 
   // 
   // 
   // ▂▂▂▂▂▂▂▂▂▂▂▂▂▂▂▂▂▂▂▂▂▂▂▂▂▂▂▂▂▂▂▂▂▂▂▂▂▂▂▂▂▂▂▂
   // 1.1     Step operation and phases
   // 
   // 
   //  ┌─────┐  The sequence progresses from one step to the next if the
   //  │Step n        │  transition logic for the step is TRUE. 
   //  └┬────┘                                                                 
   //   │       In this example, STEP n is active and will remain active
   //         --- T n        until its associated transition (T n) becomes TRUE; at this
   //   │       point the sequence will advance to the next step (STEP n+1)
   //  ┌┴────┐  and execute the actions required of this step. The sequence
   //  │Step n+1    │  will remain in this step until its transition condition is
   //  └┬────┘  true, at which point the sequence will advance again.
   //   │                                                                      
   //         --- T n+1      Each step has a step number, this is an integer value in
   //   │       the range 0 to 29999; step numbers are assigned in specific
   //           Ranges for different operating states of the sequence (IDLE,
   //           STARTING, RUNNING &c.).
   // 
   // Within an individual step, the step has three distinct phases and actions can 
   // be attached to any of these phases (externally to the block). The phases are:
   // 
   // INITIALISING (Phs_INIT)                   ┌──────┐
   // This is activated for a single OB1 scan when the step   │INITIALISING   │
   // is first processed (I.e. on the rising edge of the step     └┬─────┘
   // becoming active).                     │      
   //                           ┌┴─────┐ 
   // PROCESSING (Phs_PROC)               │PROCESSING │
   // This is the main phase of the step, it is activated        └┬─────┘
   // immediately following the INITIALISING phase and remains  │       
   // active until the step TRANSITION condition is TRUE. The     --- T n   
   // PROCESSING phase becomes inactive on the rising edge   │     
   // of the TRANSITION condition.              ┌┴─────┐
   //                           │TERMINATING │    
   // TERMINATING (Phs_TERM)               └──────┘    
   // The TERMINATING phase is activated on the rising edge of the TRANSITION
   // condition (the same condition that terminates the PROCESSING phase). The
   // terminating phase is active for a single OB1 scan.
   // 
   // 
   // [ALTERNATIVE]
   //  ┌──────┐ INITIALISING (Phs_INIT)
   //  │INITIALISING   │ This is activated for a single OB1 scan when the step
   //  └┬─────┘ is first processed (I.e. on the rising edge of the step
   //   │       becoming active).
   //  ┌┴─────┐    
   //  │PROCESSING │ PROCESSING (Phs_PROC)
   //  └┬─────┘ This is the main phase of the step, it is activated 
   //   │       immediately following the INITIALISING phase and remains
   //          --- T n       active until the step TRANSITION condition is TRUE. The
   //   │       PROCESSING phase becomes inactive on the rising edge
   //  ┌┴─────┐ of the TRANSITION condition.
   //  │TERMINATING │    
   //  └──────┘
   // 
   // TERMINATING (Phs_TERM)
   // The TERMINATING phase is activated on the rising edge of the TRANSITION
   // condition (the same condition that terminates the PROCESSING phase). The
   // terminating phase is active for a single OB1 scan.
   // 
   // 
   // 
   // 
   // ▌▌▌▌▌▌▌▌▌▌▌▌▌▌▌▌▌   GRAPHICAL FIGURE   ▐▐▐▐▐▐▐▐▐▐▐▐▐▐▐▐▐
   // 
   //     No. of scans from start of STEP 1
   //     1      2      3     4      5     6       7      8      9
   //   ┼─┼─┼─┼─┼─┼─┼─┼─┼─┼─┼─┼  ─ ─ ┐
   //                                │
   //   ┌─┐                          │
   //   │ │               Phs_INIT
   //  ─┘ └────────────────────                   
   //   ┼─┼─┼─┼─┼─┼─┼─┼─┼─┼─┼─┼                   
   //  
   //     ┌───┐                       S
   //     │   │           Phs_PROC      T
   //  ───┘   └────────────────       E
   //   ┼─┼─┼─┼─┼─┼─┼─┼─┼─┼─┼─┼       P
   //  
   //         ┌─┐                     1
   //         │ │         TRANSITION
   //  ───────┘ └──────────────
   //   ┼─┼─┼─┼─┼─┼─┼─┼─┼─┼─┼─┼
   // 
   //         ┌─┐
   //         │ │         Phs_TERM      │
   //  ───────┘ └──────────────      │
   //   ┼─┼─┼─┼─┼─┼─┼─┼─┼─┼─┼─┼  ─ ─ ┘
   // 
   // 
   //     1      2      3     4      5     6       7      8      9
   //   ┼─┼─┼─┼─┼─┼─┼─┼─┼─┼─┼─┼  ─ ─ ┐
   //                                │
   //           ┌─┐                  │
   //           │ │       Phs_INIT
   //   ────────┘ └────────────                   
   //   ┼─┼─┼─┼─┼─┼─┼─┼─┼─┼─┼─┼                   
   // 
   //             ┌───┐               S
   //             │   │   Phs_PROC      T
   //  ───────────┘   └────────       E
   //   ┼─┼─┼─┼─┼─┼─┼─┼─┼─┼─┼─┼       P
   //                           
   //                 ┌─┐             2
   //                 │ │ TRANSITION
   //  ───────────────┘ └──────      
   //   ┼─┼─┼─┼─┼─┼─┼─┼─┼─┼─┼─┼
   // 
   //                 ┌─┐
   //                 │ │ Phs_TERM      │
   //  ───────────────┘ └──────      │
   //   ┼─┼─┼─┼─┼─┼─┼─┼─┼─┼─┼─┼  ─ ─ ┘
   // 
   // 
   // 
   // ▌▌▌▌▌▌▌▌▌▌▌▌▌▌▌▌▌▌    PAL LOGO    ▐▐▐▐▐▐▐▐▐▐▐▐▐▐▐▐▐▐
   // 
   //          ⠀⠀⠀⠀⠀⠀⠀⠀⠀⠀⠀⠀⠀⠀⠀⠀⠀⠀⠀⠀⠀⠀⠀⠀⠀⠀⠀⠀⠀⣀⣀⣀
   //       ⠀⠀⠀⠀⠀⠀⠀⠀⠀⠀⠀⠀⠀⠀⠀⠀⠀⠀⠀⠀⠀⠀⠀⠀⠀⠀⠀⣤⣶⣿⣿⣿⣿⣿⣿⣤
   //       ⠀⠀⠀⠀⠀⠀⠀⠀⠀⠀⠀⠀⠀⠀⠀⠀⠀⠀⠀⠀⠀⠀⠀⠀⠀⠀⣶⣿⣿⣿⣿⣿⣿⣿⣿⣿⣶
   //       ⠀⠀⠀⠀⠀⠀⠀⠀⠀⠀⠀⠀⠀⠀⠀⠀⠀⠀⠀⠀⠀⠀⠀⠀⠀⠀⣿⣿⣿⣿⣿⣿⣿⣿⣿⣿⣿
   //       ⠀⠀⠀⠀⠀⠀⠀⠀⠀⠀⠀⠀⠀⠀⠀⠀⠀⠀⠀⠀⠀⠀⠀⠀⠀⣀⠛⣿⣿⣿⣿⣿⣿⣿⣿⣿⠿
   //       ⠀⠀⠀⠀⠀⠀⠀⠀⠀⠀⠀⠀⠀⠀⠀⠀⠀⠀⠀⠀⠀⠀⣀⣶⣿⣿⣤⠉⠿⣿⣿⣿⣿⣿⠿⠛⣤⣶
   //       ⠀⠀⠀⠀⠀⠀⠀⠀⠀⠀⠀⠀⠀⠀⠀⠀⠀⠀⠀⠀⣤⣿⣿⣿⣿⣿⣿⣿⣶⣤⠉⠉⠉⠀⠤⣿⣿⣿⣿⣶⣀⣀⣀⣀⣀⣀⣀⣀
   //       ⠀⠀⠀⠀⠀⠀⠀⠀⠀⠀⠀⠀⠀⠀⠀⠀⠀⣀⣶⣿⣿⣿⣿⣿⣿⣿⣿⣿⣿⠉⠀⠀⠀⠀⠀⠉⠿⣿⣿⣿⣿⣿⣿⣿⣿⣿⣿⣿⣶
   //       ⠀⠀⠀⠀⠀⠀⠀⠀⠀⠀⠀⠀⠀⠀⠀⠀⠛⠿⣿⣿⣿⣿⣿⣿⣿⣿⣿⠿⠀⠀⠀⠀⠀⠀⠀⠀⠀⣿⣿⣿⣿⣿⣿⣿⣿⠿⠿⣿⣿⣤
   //       ⠀⠀⠀⠀⠀⠀⠀⠀⠀⣀⣤⣶⣿⣿⣿⣿⣶⣶⣤⠉⠿⣿⣿⣿⣿⣿⠛⠀⠀⠀⠀⠀⠀⠀⠀⠀⠀⣿⣿⣿⣿⠉⠀⠀⠀⠀⠀⠉⣿⣿⣤
   //       ⠀⠀⠀⠀⠀⠀⠀⣀⣶⣿⣿⣿⣿⣿⣿⣿⣿⣿⣿⣿⣤⠉⣿⣿⣿⠛⠀⠀⠀⠀⠀⠀⠀⠀⠀⠀⣿⣿⣿⣿⣿⠀⠀⠀⠀⠀⠀⠀⠀⠿⠿
   //       ⠀⠀⠀⠀⠀⠀⣀⣿⣿⣿⣿⣿⣿⣿⣿⣿⣿⣿⣿⣿⣿⣿⠀⣿⠉⠀⠀⠀⠀⠀⠀⠀⠀⠀⠀⠀⣿⣿⣿⣿⣿
   //       ⠀⠀⠀⠀⠀⠀⣿⣿⣿⣿⣿⣿⣿⣿⣿⣿⣿⣿⣿⣿⣿⣿⣀⠀⠀⠀⠀⠀⠀⠀⠀⠀⠀⠀⠀⠀⠉⠛⠿⣿⣿⣿⣤
   //       ⠀⠀⠀⠀⠀⠀⣿⣿⣿⣿⣿⣿⣿⣿⣿⣿⣿⣿⣿⣿⣿⣿⠿⠀⠀⠀⠀⠀⠀⠀⠀⠀⠀⠀⠀⠀⠀⠀⠀⠀⠉⠛⠿⣿
   //       ⠀⠀⠀⠀⠀⠀⠛⣿⣿⣿⣿⣿⣿⣿⣿⣿⣿⣿⣿⣿⣿⣿
   //       ⠀⠀⠀⠀⠀⠀⠀⠛⣿⣿⣿⣿⣿⣿⣿⣿⣿⣿⣿⣿⠿⠉
   //       ⠀⠀⠀⠀⠀⠀⠀⠀⠀⠛⠿⣿⣿⣿⣿⣿⣿⣿⠿⠉
   //       ⠀⠀⠀⠀⠀⠀⠀⠀⠀⠀⠀⣀⣉⣉⣉⣉⣉⣀
   //       ⠀⠀⠀⠀⠀⠀⠀⠀⠀⣤⣿⣿⣿⣿⣿⣿⣿⣿⣀⠛⣿⣿⣿⣿⣿⣿⣿⣿⣿⣿⣿⣿⣿⣿⣿⣿⣿⣿⣿⣿⣿⣿⣿⣿⣿⣿⣿⣿⣿⣶⣤⣀⠀⠀⠀⠀
   //       ⠀⠀⠀⠀⠀⠀⠀⠀⣤⣿⣿⣿⠿⠉⠉⣿⣿⣿⣿⣤⠉⠿⠿⠿⠿⠿⠿⠿⠿⠿⠿⠿⠿⠿⠿⠿⠿⠿⠿⠿⠿⠿⠿⠿⠿⠿⠿⣿⣿⣿⣿⣿⣿⣀⠀⠀
   //       ⠀⠀⠀⠀⠀⠀⠀⣶⣿⣿⣿⠛⠀⠀   ⠀⠀⠿⣿⣿⣿⣤⠀⠀⠀⠀⠀⠀⣶⣶⣶⣶⣤⠀⠀⠀⠀ ⣶⣶⣶         ⣶⣶⠀⠀⠀⠀⠀⠿⣿⣿⣿⣿⣶⠀
   //       ⠀⠀⠀⠀⠀⠀⣿⣿⣿⣿⠛⠀⠀⠀⠀   ⠀⠀⠛⣿⣿⣿⣶⠀⠀⠀⠀⠀⣿⣿⣿⠿⣿⣿⠀⠀⣤⣿⣿⣿⣤       ⣿⣿⠀⠀⠀⠀⠀⠀ ⠿⣿⣿⣿⣿⣤
   //       ⠀⠀⠀⠀⠀⣿⣿⣿⣿⠉⠀⠀⠀⠀⠀   ⠀⠀⠀⠛⣿⣿⣿⣿⠀⠀⠀⠀⣿⣿⣿⣶⣿⣿⠀⠀⣿⣿⠉⣿⣿       ⣿⣿⠀⠀⠀⠀⠀     ⣿⣿⣿⣿⣿
   //       ⠀⠀⠀⣀⣿⣿⣿⣿⠉⠀⠀⠀⠀⠀⠀⠀⠀   ⠀⠀⠉⣿⣿⣿⣿      ⣿⣿⣿⠛⠛⠀⠀⣶⣿⣿⣿⣿⣿⣶    ⣿⣿⣤⣤⣤      ⣶⣿⣿⣿⣿⠛
   //       ⠀⠀⣤⣿⣿⣿⣿⠉⠀⠀⠀⠀⠀⠀⠀⠀⠀⠀⠀   ⠀⠉⣿⣿⣿⣿⣀ ⠿⠿⠿⠀⠀⠀   ⠿⠿⠉⠉⠉⠿⠿    ⠿⠿⠿⠿⠿ ⠀⣶⣿⣿⣿⣿⠿⠀
   //       ⠀⣤⣿⣿⣿⣿⣿⣶⣤⣤⣤⣤⣤⣤⣤⣤⣤⣤⣤⣤⣶⣿⣿⣿⣿⣿⣀⠀⣶⣶⣶⣶⣶⣶⣶⣶⣶⣶⣶⣶⣶⣶⣶⣶⣶⣶⣶⣶⣿⣿⣿⣿⠉⠀⠀
   //       ⠀⣿⣿⣿⣿⣿⣿⣿⣿⣿⣿⣿⣿⣿⣿⣿⣿⣿⣿⣿⣿⣿⣿⣿⣿⣿⣿⠀⠉⣿⣿⣿⣿⣿⣿⣿⣿⣿⣿⣿⣿⣿⣿⣿⣿⣿⣿⣿⣿⠿⠛⠉⠀⠀⠀⠀
   //       ⠀⠉⠛⠛⠛⠛⠛⠛⠛⠛⠛⠛⠛⠛⠛⠛⠛⠛⠛⠛⠛⠛⠛⠛⠛⠛⠉⠀⠀⠉⠉⠉⠉⠉⠉⠉⠉⠉⠉⠉⠉⠉⠉⠉⠉⠉⠉⠉⠀⠀⠀⠀⠀⠀⠀⠀
   // ↳
   //                ━━━   ⬙⬙⬙⬙⬙⬙   ━━━
   // ↳
   // ↳
   // ██████████████ █ █ █ █  END   █ █ █ █ ██████████████
   // ↳
END_REGION

REGION Network 12: Special characters — Hyphens, whitespace and construction lines
   // ▀▀▀▀▀▀▀▀▀▀▀▀▀▀▀▀▀▀▀▀▀▀▀▀▀▀▀▀▀▀▀▀▀▀▀▀▀▀▀▀▀▀▀▀
   // 
   // TITLE:    SPECIAL CHARACTERS
   // 
   // ▄▄▄▄▄▄▄▄▄▄▄▄▄▄▄▄▄▄▄▄▄▄▄▄▄▄▄▄▄▄▄▄▄▄▄▄▄▄▄▄▄▄▄▄
   // 
   // 
   // The TIA Portal Basic font contains many different types of characters:
   // 
   //    •   Hyphens and whitespace characters
   //    •   Construction lines (these are specially ordered characters, useful for building tables &c.)
   //    •   Arrows
   //    •   Box characters (for drawing box and line diagrams)
   //    •   Block characters
   //    •   Currency
   //    •   Punctuation (extended list)
   //    •   Non-proportional letters and numbers
   //    •   Greek characters
   //    •   Indexing characters
   //    •   Roman numerals
   //    •   Mathematical characters
   //    •   Geometric characters
   //    •   Dingbat characters
   // 
   // The following sections contain a list of these characters for use in TIA Portal comment fields.
   // 
   // Note:    The following tables of characters break the rules for comment fields by exceeding
   //      the prescribed comment field width of 44 em-spaces. This is done to give the 
   //      characters in a more concise form whilst maintaining reasonable descriptions for
   //      the characters
   // 
   // 
   // 
   // ▄▄▄▄▄▄▄▄▄▄▄▄▄▄▄▄▄▄▄▄▄▄▄▄▄▄▄▄▄▄▄▄▄▄▄▄▄▄▄▄▄▄▄▄
   // HYPHENS AND WHITESPACE CHARACTERS
   // 
   // 
   // — Em Dash               █ █ Em Space
   // –   En Dash              █ █   En Space
   // ‐    Hyphen               █ █    Three-Per-Em Space
   // ¬   Soft Hyphen             █ █    Normal Space
   //                       █ █     Six-Per-Em Space
   // 
   // 
   // 
   // ▄▄▄▄▄▄▄▄▄▄▄▄▄▄▄▄▄▄▄▄▄▄▄▄▄▄▄▄▄▄▄▄▄▄▄▄▄▄▄▄▄▄▄▄
   // CONSTRUCTION LINES AND USEFUL LINES
   // 
   // 
   // [Copyable whitespace]
   //  █ █ █ █ █ Em En ThreePerEm SixPerEM
   // [Em-space construction line]
   // ▀▄▀▄▀▄▀▄▀▄▀▄▀▄▀▄▀▄▀▄▀▄▀▄▀▄▀▄▀▄▀▄▀▄▀▄▀▄▀▄▀▄▀▄
   // [Central header — used for examples]
   // ▌▌▌▌▌▌▌▌▌▌▌▌▌▌▌▌▌▌▌▌▌▌▐▐▐▐▐▐▐▐▐▐▐▐▐▐▐▐▐▐▐▐▐▐
   // [Title start]
   // ▀▀▀▀▀▀▀▀▀▀▀▀▀▀▀▀▀▀▀▀▀▀▀▀▀▀▀▀▀▀▀▀▀▀▀▀▀▀▀▀▀▀▀▀
   // [Title end/section over-line]
   // ▄▄▄▄▄▄▄▄▄▄▄▄▄▄▄▄▄▄▄▄▄▄▄▄▄▄▄▄▄▄▄▄▄▄▄▄▄▄▄▄▄▄▄▄
   // [Subsection over-line]
   // ▂▂▂▂▂▂▂▂▂▂▂▂▂▂▂▂▂▂▂▂▂▂▂▂▂▂▂▂▂▂▂▂▂▂▂▂▂▂▂▂▂▂▂▂
   // [Inline section over-line]
   // ▁▁▁▁▁▁▁▁▁▁▁▁▁▁▁▁▁▁▁▁▁▁▁▁▁▁▁▁▁▁▁▁▁▁▁▁▁▁▁▁▁▁▁▁
   // [Table row line]
   //  ――――――――――――――――――――――――――――――――――――――――――
   // [Revision row line]
   //  ―――――――――――――――――――――――――――――――――――――――――――
   // [Flourish divider]
   //                ━━━   ⬙⬙⬙⬙⬙⬙   ━━━
   // [End line]
   // ██████████████ █ █ █ █  END   █ █ █ █ ██████████████
END_REGION

